  MoveL 2642 to (274.37, 10.03, -264.36) mm, rotated rx -179.9 ry 0 rz -90 deg; joints [33.189, -61.203, 97.914, -131.675, 47.114, 143.425]
  MoveC 2643 to (277.1, 10.02, -263.23) mm, rotated rx -179.9 ry 0 rz -90 deg; joints [33.299, -61.17, 97.861, -131.541, 47.167, 143.324] to (278.23, 10.02, -260.51) mm, rotated rx -179.9 ry 0 rz -90 deg; joints [33.393, -61.271, 98.014, -131.475, 47.257, 143.309]
  MoveL 2644 to (278.23, 10.02, -260.51) mm, rotated rx -179.9 ry 0 rz -90 deg; joints [33.393, -61.271, 98.014, -131.475, 47.257, 143.309]
  MoveL 2645 to (278.23, 10.03, -85.81) mm, rotated rx -179.9 ry 0 rz -90 deg; joints [37.456, -69.808, 110.438, -129.685, 52.193, 144.471]
  MoveC 2646 to (276.95, 10.02, -81.59) mm, rotated rx -179.9 ry 0 rz -90 deg; joints [37.521, -70.054, 110.778, -129.674, 52.292, 144.523] to (273.55, 10.03, -78.79) mm, rotated rx -179.9 ry 0 rz -90 deg; joints [37.48, -70.309, 111.133, -129.777, 52.332, 144.646]
  MoveL 2647 to (273.55, 10.02, -78.79) mm, rotated rx -179.9 ry 0 rz -90 deg; joints [37.48, -70.309, 111.133, -129.777, 52.332, 144.646]
  MoveC 2648 to (270.14, 10.02, -75.98) mm, rotated rx -179.9 ry 0 rz -90 deg; joints [37.438, -70.563, 111.486, -129.878, 52.371, 144.767] to (268.86, 10.02, -71.76) mm, rotated rx -179.9 ry 0 rz -90 deg; joints [37.504, -70.809, 111.823, -129.864, 52.468, 144.816]
  MoveL 2649 to (268.86, 10.02, -71.76) mm, rotated rx -179.9 ry 0 rz -90 deg; joints [37.504, -70.809, 111.823, -129.864, 52.468, 144.816]
  MoveL 2650 to (268.86, 10.02, -61.09) mm, rotated rx -179.9 ry 0 rz -90 deg; joints [37.783, -71.313, 112.509, -129.684, 52.746, 144.821]
  MoveC 2651 to (267.74, 10.03, -58.37) mm, rotated rx -179.9 ry 0 rz -90 deg; joints [37.817, -71.483, 112.74, -129.685, 52.804, 144.86] to (265.01, 10.02, -57.24) mm, rotated rx -179.9 ry 0 rz -90 deg; joints [37.754, -71.635, 112.948, -129.783, 52.804, 144.953]
  MoveL 2652 to (265.01, 10.02, -57.24) mm, rotated rx -179.9 ry 0 rz -90 deg; joints [37.754, -71.635, 112.948, -129.783, 52.804, 144.953]
  MoveL 2653 to (-265.01, 10.02, -57.24) mm, rotated rx -179.9 ry 0 rz -90 deg; joints [15.13, -86.315, 131.2, -158.711, 45.944, 165.304]
  MoveC 2654 to (-267.74, 10.03, -58.37) mm, rotated rx -179.9 ry 0 rz -90 deg; joints [14.976, -86.289, 131.174, -158.919, 45.905, 165.446] to (-268.86, 10.02, -61.09) mm, rotated rx -179.9 ry 0 rz -90 deg; joints [14.882, -86.136, 131.013, -159.043, 45.873, 165.528]
  MoveL 2655 to (-268.86, 10.03, -61.09) mm, rotated rx -179.9 ry 0 rz -90 deg; joints [14.882, -86.136, 131.013, -159.043, 45.873, 165.528]
  MoveL 2656 to (-268.86, 10.02, -251.14) mm, rotated rx -179.9 ry 0 rz -90 deg; joints [12.675, -74.659, 117.443, -161.372, 43.366, 166.653]
  MoveC 2657 to (-267.74, 10.02, -253.87) mm, rotated rx -179.9 ry 0 rz -90 deg; joints [12.698, -74.485, 117.216, -161.322, 43.321, 166.605] to (-265.01, 10.02, -255) mm, rotated rx -179.9 ry 0 rz -90 deg; joints [12.805, -74.383, 117.082, -161.158, 43.316, 166.481]
  MoveL 2658 to (-265.01, 10.03, -255) mm, rotated rx -179.9 ry 0 rz -90 deg; joints [12.805, -74.383, 117.082, -161.158, 43.316, 166.481]
  MoveL 2659 to (265.01, 10.02, -255) mm, rotated rx -179.9 ry 0 rz -90 deg; joints [33.086, -61.986, 99.114, -132.076, 47.331, 143.923]
  MoveC 2660 to (267.74, 10.02, -253.87) mm, rotated rx -179.9 ry 0 rz -90 deg; joints [33.197, -61.954, 99.063, -131.941, 47.384, 143.823] to (268.86, 10.02, -251.14) mm, rotated rx -179.9 ry 0 rz -90 deg; joints [33.291, -62.054, 99.214, -131.873, 47.474, 143.806]
  MoveL 2661 to (268.86, 10.02, -251.14) mm, rotated rx -179.9 ry 0 rz -90 deg; joints [33.291, -62.054, 99.214, -131.873, 47.474, 143.806]
  MoveL 2662 to (268.86, 10.02, -71.76) mm, rotated rx -179.9 ry 0 rz -90 deg; joints [37.504, -70.809, 111.823, -129.864, 52.468, 144.816]
  MoveC 2663 to (266.09, 10.02, -66.2) mm, rotated rx -179.9 ry 0 rz -90 deg; joints [37.555, -71.172, 112.321, -129.89, 52.584, 144.914] to (259.98, 10.02, -65.06) mm, rotated rx -179.9 ry 0 rz -90 deg; joints [37.377, -71.445, 112.699, -130.135, 52.548, 145.124]
  MoveL 2664 to (259.98, 10.03, -65.06) mm, rotated rx -179.9 ry 0 rz -90 deg; joints [37.377, -71.445, 112.699, -130.135, 52.548, 145.124]
  MoveC 2665 to (254.53, 10.03, -66.22) mm, rotated rx -179.9 ry 0 rz -90 deg; joints [37.161, -71.585, 112.895, -130.392, 52.46, 145.31] to (248.97, 10.03, -66.6) mm, rotated rx -179.9 ry 0 rz -90 deg; joints [36.959, -71.764, 113.144, -130.641, 52.391, 145.501]
  MoveL 2666 to (248.97, 10.02, -66.6) mm, rotated rx -179.9 ry 0 rz -90 deg; joints [36.959, -71.764, 113.144, -130.641, 52.391, 145.501]
  MoveL 2667 to (-255.65, 10.03, -66.6) mm, rotated rx -179.9 ry 0 rz -90 deg; joints [15.473, -85.568, 130.397, -158.231, 45.981, 164.961]
  MoveC 2668 to (-258.37, 10.03, -67.73) mm, rotated rx -179.9 ry 0 rz -90 deg; joints [15.321, -85.544, 130.373, -158.436, 45.941, 165.101] to (-259.5, 10.03, -70.46) mm, rotated rx -179.9 ry 0 rz -90 deg; joints [15.226, -85.393, 130.211, -158.559, 45.907, 165.182]
  MoveL 2669 to (-259.5, 10.03, -70.46) mm, rotated rx -179.9 ry 0 rz -90 deg; joints [15.226, -85.393, 130.211, -158.559, 45.907, 165.182]
  MoveL 2670 to (-259.5, 10.03, -241.78) mm, rotated rx -179.9 ry 0 rz -90 deg; joints [13.181, -75.083, 117.987, -160.698, 43.599, 166.199]
  MoveC 2671 to (-258.37, 10.02, -244.5) mm, rotated rx -179.9 ry 0 rz -90 deg; joints [13.203, -74.908, 117.76, -160.65, 43.555, 166.153] to (-255.65, 10.03, -245.63) mm, rotated rx -179.9 ry 0 rz -90 deg; joints [13.31, -74.805, 117.625, -160.488, 43.551, 166.029]
  MoveL 2672 to (-255.65, 10.02, -245.63) mm, rotated rx -179.9 ry 0 rz -90 deg; joints [13.31, -74.805, 117.625, -160.488, 43.551, 166.029]
  MoveL 2673 to (255.65, 10.03, -245.63) mm, rotated rx -179.9 ry 0 rz -90 deg; joints [32.98, -62.765, 100.3, -132.467, 47.543, 144.407]
  MoveC 2674 to (258.37, 10.03, -244.5) mm, rotated rx -179.9 ry 0 rz -90 deg; joints [33.093, -62.734, 100.25, -132.331, 47.596, 144.307] to (259.5, 10.03, -241.78) mm, rotated rx -179.9 ry 0 rz -90 deg; joints [33.187, -62.834, 100.4, -132.261, 47.684, 144.288]
  MoveL 2675 to (259.5, 10.02, -241.78) mm, rotated rx -179.9 ry 0 rz -90 deg; joints [33.187, -62.834, 100.4, -132.261, 47.684, 144.288]
  MoveL 2676 to (259.5, 10.03, -70.46) mm, rotated rx -179.9 ry 0 rz -90 deg; joints [37.22, -71.206, 112.375, -130.248, 52.404, 145.139]
  MoveC 2677 to (258.37, 10.03, -67.73) mm, rotated rx -179.9 ry 0 rz -90 deg; joints [37.253, -71.376, 112.607, -130.251, 52.462, 145.178] to (255.65, 10.02, -66.6) mm, rotated rx -179.9 ry 0 rz -90 deg; joints [37.189, -71.527, 112.815, -130.35, 52.462, 145.272]
  MoveL 2678 to (255.65, 10.03, -66.6) mm, rotated rx -179.9 ry 0 rz -90 deg; joints [37.189, -71.527, 112.815, -130.35, 52.462, 145.272]
  MoveL 2679 to (248.97, 10.02, -66.6) mm, rotated rx -179.9 ry 0 rz -90 deg; joints [36.959, -71.764, 113.144, -130.641, 52.391, 145.501]
  MoveC 2680 to (244.46, 10.03, -67.86) mm, rotated rx -179.9 ry 0 rz -90 deg; joints [36.771, -71.864, 113.283, -130.86, 52.31, 145.656] to (241.27, 10.02, -71.28) mm, rotated rx -179.9 ry 0 rz -90 deg; joints [36.572, -71.812, 113.218, -131.059, 52.188, 145.766]
  MoveL 2681 to (241.27, 10.02, -71.28) mm, rotated rx -179.9 ry 0 rz -90 deg; joints [36.572, -71.812, 113.218, -131.059, 52.188, 145.766]
  MoveC 2682 to (238.08, 10.03, -74.7) mm, rotated rx -179.9 ry 0 rz -90 deg; joints [36.374, -71.76, 113.151, -131.258, 52.067, 145.877] to (233.58, 10.02, -75.96) mm, rotated rx -179.9 ry 0 rz -90 deg; joints [36.185, -71.856, 113.287, -131.479, 51.986, 146.033]
  MoveL 2683 to (233.58, 10.03, -75.96) mm, rotated rx -179.9 ry 0 rz -90 deg; joints [36.185, -71.856, 113.287, -131.479, 51.986, 146.033]
  MoveL 2684 to (-246.29, 10.03, -75.96) mm, rotated rx -179.9 ry 0 rz -90 deg; joints [15.809, -84.825, 129.586, -157.757, 46.008, 164.619]
  MoveC 2685 to (-249.01, 10.02, -77.09) mm, rotated rx -179.9 ry 0 rz -90 deg; joints [15.658, -84.802, 129.563, -157.959, 45.967, 164.757] to (-250.14, 10.03, -79.82) mm, rotated rx -179.9 ry 0 rz -90 deg; joints [15.564, -84.652, 129.401, -158.081, 45.93, 164.836]
  MoveL 2686 to (-250.14, 10.02, -79.82) mm, rotated rx -179.9 ry 0 rz -90 deg; joints [15.564, -84.652, 129.401, -158.081, 45.93, 164.836]
  MoveL 2687 to (-250.14, 10.02, -232.42) mm, rotated rx -179.9 ry 0 rz -90 deg; joints [13.693, -75.502, 118.519, -160.021, 43.832, 165.744]
  MoveC 2688 to (-249.01, 10.02, -235.14) mm, rotated rx -179.9 ry 0 rz -90 deg; joints [13.713, -75.326, 118.294, -159.975, 43.79, 165.699] to (-246.29, 10.02, -236.27) mm, rotated rx -179.9 ry 0 rz -90 deg; joints [13.821, -75.222, 118.158, -159.813, 43.787, 165.577]
  MoveL 2689 to (-246.29, 10.02, -236.27) mm, rotated rx -179.9 ry 0 rz -90 deg; joints [13.821, -75.222, 118.158, -159.813, 43.787, 165.577]
  MoveL 2690 to (246.29, 10.03, -236.27) mm, rotated rx -179.9 ry 0 rz -90 deg; joints [32.873, -63.542, 101.472, -132.85, 47.748, 144.878]
  MoveC 2691 to (249.01, 10.03, -235.14) mm, rotated rx -179.9 ry 0 rz -90 deg; joints [32.987, -63.511, 101.423, -132.713, 47.801, 144.778] to (250.14, 10.03, -232.42) mm, rotated rx -179.9 ry 0 rz -90 deg; joints [33.082, -63.612, 101.571, -132.641, 47.889, 144.757]
  MoveL 2692 to (250.14, 10.03, -232.42) mm, rotated rx -179.9 ry 0 rz -90 deg; joints [33.082, -63.612, 101.571, -132.641, 47.889, 144.757]
  MoveL 2693 to (250.14, 10.03, -79.82) mm, rotated rx -179.9 ry 0 rz -90 deg; joints [36.659, -71.091, 112.231, -130.813, 52.063, 145.458]
  MoveC 2694 to (249.01, 10.03, -77.09) mm, rotated rx -179.9 ry 0 rz -90 deg; joints [36.69, -71.261, 112.464, -130.817, 52.122, 145.499] to (246.29, 10.02, -75.96) mm, rotated rx -179.9 ry 0 rz -90 deg; joints [36.625, -71.411, 112.67, -130.918, 52.122, 145.593]
  MoveL 2695 to (246.29, 10.02, -75.96) mm, rotated rx -179.9 ry 0 rz -90 deg; joints [36.625, -71.411, 112.67, -130.918, 52.122, 145.593]
  MoveL 2696 to (233.58, 10.03, -75.96) mm, rotated rx -179.9 ry 0 rz -90 deg; joints [36.185, -71.856, 113.287, -131.479, 51.986, 146.033]
  MoveC 2697 to (229.36, 10.02, -77.24) mm, rotated rx -179.9 ry 0 rz -90 deg; joints [36.005, -71.941, 113.406, -131.689, 51.908, 146.179] to (226.56, 10.02, -80.65) mm, rotated rx -179.9 ry 0 rz -90 deg; joints [35.82, -71.873, 113.318, -131.872, 51.792, 146.278]
  MoveL 2698 to (226.56, 10.02, -80.65) mm, rotated rx -179.9 ry 0 rz -90 deg; joints [35.82, -71.873, 113.318, -131.872, 51.792, 146.278]
  MoveC 2699 to (223.75, 10.02, -84.05) mm, rotated rx -179.9 ry 0 rz -90 deg; joints [35.636, -71.805, 113.23, -132.055, 51.676, 146.376] to (219.54, 10.03, -85.33) mm, rotated rx -179.9 ry 0 rz -90 deg; joints [35.455, -71.888, 113.346, -132.266, 51.598, 146.524]
  MoveL 2700 to (219.54, 10.03, -85.33) mm, rotated rx -179.9 ry 0 rz -90 deg; joints [35.455, -71.888, 113.346, -132.266, 51.598, 146.524]
  MoveL 2701 to (-236.92, 10.03, -85.33) mm, rotated rx -179.9 ry 0 rz -90 deg; joints [16.137, -84.084, 128.767, -157.288, 46.024, 164.277]
  MoveC 2702 to (-239.65, 10.03, -86.46) mm, rotated rx -179.9 ry 0 rz -90 deg; joints [15.988, -84.063, 128.745, -157.488, 45.983, 164.413] to (-240.78, 10.02, -89.18) mm, rotated rx -179.9 ry 0 rz -90 deg; joints [15.894, -83.915, 128.582, -157.608, 45.944, 164.491]
  MoveL 2703 to (-240.78, 10.02, -89.18) mm, rotated rx -179.9 ry 0 rz -90 deg; joints [15.894, -83.915, 128.582, -157.608, 45.944, 164.491]
  MoveL 2704 to (-240.78, 10.02, -223.05) mm, rotated rx -179.9 ry 0 rz -90 deg; joints [14.21, -75.915, 119.042, -159.339, 44.065, 165.288]
  MoveC 2705 to (-239.65, 10.03, -225.78) mm, rotated rx -179.9 ry 0 rz -90 deg; joints [14.229, -75.739, 118.817, -159.295, 44.024, 165.244] to (-236.92, 10.02, -226.91) mm, rotated rx -179.9 ry 0 rz -90 deg; joints [14.337, -75.634, 118.68, -159.134, 44.023, 165.123]
  MoveL 2706 to (-236.92, 10.02, -226.91) mm, rotated rx -179.9 ry 0 rz -90 deg; joints [14.337, -75.634, 118.68, -159.134, 44.023, 165.123]
  MoveL 2707 to (236.92, 10.02, -226.91) mm, rotated rx -179.9 ry 0 rz -90 deg; joints [32.764, -64.316, 102.631, -133.225, 47.948, 145.336]
  MoveC 2708 to (239.65, 10.02, -225.78) mm, rotated rx -179.9 ry 0 rz -90 deg; joints [32.879, -64.285, 102.582, -133.087, 48.001, 145.236] to (240.78, 10.02, -223.05) mm, rotated rx -179.9 ry 0 rz -90 deg; joints [32.975, -64.386, 102.73, -133.012, 48.088, 145.213]
  MoveL 2709 to (240.78, 10.02, -223.05) mm, rotated rx -179.9 ry 0 rz -90 deg; joints [32.975, -64.386, 102.73, -133.012, 48.088, 145.213]
  MoveL 2710 to (240.78, 10.02, -89.18) mm, rotated rx -179.9 ry 0 rz -90 deg; joints [36.098, -70.969, 112.076, -131.38, 51.724, 145.78]
  MoveC 2711 to (239.65, 10.03, -86.46) mm, rotated rx -179.9 ry 0 rz -90 deg; joints [36.128, -71.139, 112.31, -131.386, 51.783, 145.821] to (236.92, 10.02, -85.33) mm, rotated rx -179.9 ry 0 rz -90 deg; joints [36.063, -71.288, 112.515, -131.488, 51.783, 145.916]
  MoveL 2712 to (236.92, 10.02, -85.33) mm, rotated rx -179.9 ry 0 rz -90 deg; joints [36.063, -71.288, 112.515, -131.488, 51.783, 145.916]
  MoveL 2713 to (219.54, 10.03, -85.33) mm, rotated rx -179.9 ry 0 rz -90 deg; joints [35.455, -71.888, 113.346, -132.266, 51.598, 146.524]
  MoveC 2714 to (215.32, 10.02, -86.61) mm, rotated rx -179.9 ry 0 rz -90 deg; joints [35.275, -71.969, 113.461, -132.477, 51.52, 146.672] to (212.51, 10.03, -90.01) mm, rotated rx -179.9 ry 0 rz -90 deg; joints [35.091, -71.899, 113.369, -132.661, 51.405, 146.771]
  MoveL 2715 to (212.51, 10.03, -90.01) mm, rotated rx -179.9 ry 0 rz -90 deg; joints [35.091, -71.899, 113.369, -132.661, 51.405, 146.771]
  MoveC 2716 to (209.71, 10.03, -93.41) mm, rotated rx -179.9 ry 0 rz -90 deg; joints [34.907, -71.827, 113.276, -132.845, 51.289, 146.871] to (205.49, 10.02, -94.69) mm, rotated rx -179.9 ry 0 rz -90 deg; joints [34.726, -71.906, 113.388, -133.058, 51.212, 147.02]
  MoveL 2717 to (205.49, 10.02, -94.69) mm, rotated rx -179.9 ry 0 rz -90 deg; joints [34.726, -71.906, 113.388, -133.058, 51.212, 147.02]
  MoveL 2718 to (-227.56, 10.02, -94.69) mm, rotated rx -179.9 ry 0 rz -90 deg; joints [16.459, -83.347, 127.939, -156.825, 46.03, 163.935]
  MoveC 2719 to (-230.29, 10.03, -95.82) mm, rotated rx -179.9 ry 0 rz -90 deg; joints [16.311, -83.326, 127.918, -157.022, 45.988, 164.07] to (-231.41, 10.03, -98.54) mm, rotated rx -179.9 ry 0 rz -90 deg; joints [16.218, -83.18, 127.754, -157.14, 45.947, 164.146]
  MoveL 2720 to (-231.41, 10.03, -98.54) mm, rotated rx -179.9 ry 0 rz -90 deg; joints [16.218, -83.18, 127.754, -157.14, 45.947, 164.146]
  MoveL 2721 to (-231.41, 10.02, -213.69) mm, rotated rx -179.9 ry 0 rz -90 deg; joints [14.733, -76.323, 119.554, -158.654, 44.299, 164.831]
  MoveC 2722 to (-230.29, 10.02, -216.42) mm, rotated rx -179.9 ry 0 rz -90 deg; joints [14.751, -76.147, 119.33, -158.611, 44.259, 164.788] to (-227.56, 10.03, -217.54) mm, rotated rx -179.9 ry 0 rz -90 deg; joints [14.858, -76.04, 119.192, -158.451, 44.259, 164.668]
  MoveL 2723 to (-227.56, 10.03, -217.55) mm, rotated rx -179.9 ry 0 rz -90 deg; joints [14.858, -76.04, 119.192, -158.451, 44.259, 164.668]
  MoveL 2724 to (227.56, 10.02, -217.55) mm, rotated rx -179.9 ry 0 rz -90 deg; joints [32.654, -65.088, 103.776, -133.592, 48.142, 145.782]
  MoveC 2725 to (230.29, 10.02, -216.42) mm, rotated rx -179.9 ry 0 rz -90 deg; joints [32.769, -65.058, 103.729, -133.453, 48.195, 145.682] to (231.41, 10.03, -213.69) mm, rotated rx -179.9 ry 0 rz -90 deg; joints [32.866, -65.158, 103.875, -133.376, 48.281, 145.657]
  MoveL 2726 to (231.41, 10.02, -213.69) mm, rotated rx -179.9 ry 0 rz -90 deg; joints [32.866, -65.158, 103.875, -133.376, 48.281, 145.657]
  MoveL 2727 to (231.41, 10.03, -98.54) mm, rotated rx -179.9 ry 0 rz -90 deg; joints [35.54, -70.839, 111.911, -131.948, 51.386, 146.103]
  MoveC 2728 to (230.29, 10.03, -95.82) mm, rotated rx -179.9 ry 0 rz -90 deg; joints [35.569, -71.009, 112.145, -131.955, 51.444, 146.145] to (227.56, 10.03, -94.69) mm, rotated rx -179.9 ry 0 rz -90 deg; joints [35.502, -71.158, 112.35, -132.059, 51.445, 146.241]
  MoveL 2729 to (227.56, 10.03, -94.69) mm, rotated rx -179.9 ry 0 rz -90 deg; joints [35.502, -71.158, 112.35, -132.059, 51.445, 146.241]
  MoveL 2730 to (205.49, 10.02, -94.69) mm, rotated rx -179.9 ry 0 rz -90 deg; joints [34.726, -71.906, 113.388, -133.058, 51.212, 147.02]
  MoveC 2731 to (201.27, 10.02, -95.97) mm, rotated rx -179.9 ry 0 rz -90 deg; joints [34.544, -71.985, 113.499, -133.273, 51.134, 147.17] to (198.47, 10.03, -99.37) mm, rotated rx -179.9 ry 0 rz -90 deg; joints [34.361, -71.911, 113.403, -133.457, 51.019, 147.27]
  MoveL 2732 to (198.47, 10.02, -99.37) mm, rotated rx -179.9 ry 0 rz -90 deg; joints [34.361, -71.911, 113.403, -133.457, 51.019, 147.27]
  MoveC 2733 to (195.67, 10.02, -102.78) mm, rotated rx -179.9 ry 0 rz -90 deg; joints [34.177, -71.836, 113.305, -133.642, 50.904, 147.371] to (191.45, 10.02, -104.05) mm, rotated rx -179.9 ry 0 rz -90 deg; joints [33.995, -71.912, 113.413, -133.858, 50.827, 147.521]
  MoveL 2734 to (191.45, 10.02, -104.05) mm, rotated rx -179.9 ry 0 rz -90 deg; joints [33.995, -71.912, 113.413, -133.858, 50.827, 147.521]
  MoveL 2735 to (-218.2, 10.02, -104.05) mm, rotated rx -179.9 ry 0 rz -90 deg; joints [16.775, -82.612, 127.102, -156.366, 46.027, 163.592]
  MoveC 2736 to (-220.92, 10.02, -105.18) mm, rotated rx -179.9 ry 0 rz -90 deg; joints [16.628, -82.592, 127.082, -156.561, 45.984, 163.725] to (-222.05, 10.02, -107.91) mm, rotated rx -179.9 ry 0 rz -90 deg; joints [16.535, -82.448, 126.918, -156.677, 45.94, 163.8]
  MoveL 2737 to (-222.05, 10.03, -107.91) mm, rotated rx -179.9 ry 0 rz -90 deg; joints [16.535, -82.448, 126.918, -156.677, 45.94, 163.8]
  MoveL 2738 to (-222.05, 10.02, -204.33) mm, rotated rx -179.9 ry 0 rz -90 deg; joints [15.261, -76.726, 120.056, -157.964, 44.534, 164.373]
  MoveC 2739 to (-220.92, 10.03, -207.05) mm, rotated rx -179.9 ry 0 rz -90 deg; joints [15.278, -76.549, 119.833, -157.923, 44.495, 164.331] to (-218.2, 10.02, -208.18) mm, rotated rx -179.9 ry 0 rz -90 deg; joints [15.385, -76.44, 119.693, -157.765, 44.496, 164.212]
  MoveL 2740 to (-218.2, 10.03, -208.18) mm, rotated rx -179.9 ry 0 rz -90 deg; joints [15.385, -76.44, 119.693, -157.765, 44.496, 164.212]
  MoveL 2741 to (218.2, 10.03, -208.18) mm, rotated rx -179.9 ry 0 rz -90 deg; joints [32.541, -65.858, 104.909, -133.951, 48.329, 146.215]
  MoveC 2742 to (220.92, 10.02, -207.05) mm, rotated rx -179.9 ry 0 rz -90 deg; joints [32.657, -65.828, 104.863, -133.811, 48.383, 146.115] to (222.05, 10.02, -204.33) mm, rotated rx -179.9 ry 0 rz -90 deg; joints [32.755, -65.929, 105.008, -133.732, 48.468, 146.088]
  MoveL 2743 to (222.05, 10.02, -204.33) mm, rotated rx -179.9 ry 0 rz -90 deg; joints [32.755, -65.929, 105.008, -133.732, 48.468, 146.088]
  MoveL 2744 to (222.05, 10.02, -107.91) mm, rotated rx -179.9 ry 0 rz -90 deg; joints [34.983, -70.701, 111.734, -132.517, 51.049, 146.428]
  MoveC 2745 to (220.92, 10.02, -105.18) mm, rotated rx -179.9 ry 0 rz -90 deg; joints [35.011, -70.872, 111.969, -132.526, 51.107, 146.47] to (218.2, 10.02, -104.05) mm, rotated rx -179.9 ry 0 rz -90 deg; joints [34.943, -71.02, 112.173, -132.632, 51.108, 146.568]
  MoveL 2746 to (218.2, 10.02, -104.05) mm, rotated rx -179.9 ry 0 rz -90 deg; joints [34.943, -71.02, 112.173, -132.632, 51.108, 146.568]
  MoveL 2747 to (191.45, 10.02, -104.05) mm, rotated rx -179.9 ry 0 rz -90 deg; joints [33.995, -71.912, 113.413, -133.858, 50.827, 147.521]
  MoveC 2748 to (187.23, 10.03, -105.33) mm, rotated rx -179.9 ry 0 rz -90 deg; joints [33.813, -71.988, 113.519, -134.074, 50.751, 147.672] to (184.43, 10.02, -108.73) mm, rotated rx -179.9 ry 0 rz -90 deg; joints [33.63, -71.911, 113.419, -134.26, 50.636, 147.774]
  MoveL 2749 to (184.43, 10.02, -108.73) mm, rotated rx -179.9 ry 0 rz -90 deg; joints [33.63, -71.911, 113.419, -134.26, 50.636, 147.774]
  MoveC 2750 to (181.62, 10.02, -112.14) mm, rotated rx -179.9 ry 0 rz -90 deg; joints [33.448, -71.832, 113.317, -134.445, 50.522, 147.876] to (177.4, 10.02, -113.42) mm, rotated rx -179.9 ry 0 rz -90 deg; joints [33.265, -71.906, 113.42, -134.663, 50.446, 148.028]
  MoveL 2751 to (177.4, 10.02, -113.42) mm, rotated rx -179.9 ry 0 rz -90 deg; joints [33.265, -71.906, 113.42, -134.663, 50.446, 148.028]
  MoveL 2752 to (-208.84, 10.02, -113.42) mm, rotated rx -179.9 ry 0 rz -90 deg; joints [17.084, -81.879, 126.257, -155.911, 46.013, 163.249]
  MoveC 2753 to (-211.56, 10.03, -114.54) mm, rotated rx -179.9 ry 0 rz -90 deg; joints [16.938, -81.861, 126.238, -156.104, 45.97, 163.38] to (-212.69, 10.03, -117.27) mm, rotated rx -179.9 ry 0 rz -90 deg; joints [16.846, -81.718, 126.074, -156.219, 45.924, 163.453]
  MoveL 2754 to (-212.69, 10.03, -117.27) mm, rotated rx -179.9 ry 0 rz -90 deg; joints [16.846, -81.718, 126.074, -156.219, 45.924, 163.453]
  MoveL 2755 to (-212.69, 10.03, -194.97) mm, rotated rx -179.9 ry 0 rz -90 deg; joints [15.795, -77.123, 120.548, -157.271, 44.769, 163.913]
  MoveC 2756 to (-211.56, 10.02, -197.69) mm, rotated rx -179.9 ry 0 rz -90 deg; joints [15.811, -76.946, 120.325, -157.231, 44.731, 163.873] to (-208.84, 10.02, -198.82) mm, rotated rx -179.9 ry 0 rz -90 deg; joints [15.918, -76.835, 120.184, -157.074, 44.734, 163.755]
  MoveL 2757 to (-208.84, 10.03, -198.82) mm, rotated rx -179.9 ry 0 rz -90 deg; joints [15.918, -76.835, 120.184, -157.074, 44.734, 163.755]
  MoveL 2758 to (208.84, 10.03, -198.82) mm, rotated rx -179.9 ry 0 rz -90 deg; joints [32.426, -66.626, 106.03, -134.303, 48.511, 146.636]
  MoveC 2759 to (211.56, 10.02, -197.69) mm, rotated rx -179.9 ry 0 rz -90 deg; joints [32.543, -66.596, 105.984, -134.162, 48.565, 146.536] to (212.69, 10.02, -194.97) mm, rotated rx -179.9 ry 0 rz -90 deg; joints [32.641, -66.697, 106.129, -134.081, 48.649, 146.507]
  MoveL 2760 to (212.69, 10.03, -194.97) mm, rotated rx -179.9 ry 0 rz -90 deg; joints [32.641, -66.697, 106.129, -134.081, 48.649, 146.507]
  MoveL 2761 to (212.69, 10.02, -117.27) mm, rotated rx -179.9 ry 0 rz -90 deg; joints [34.429, -70.556, 111.547, -133.087, 50.713, 146.755]
  MoveC 2762 to (211.56, 10.03, -114.54) mm, rotated rx -179.9 ry 0 rz -90 deg; joints [34.455, -70.728, 111.783, -133.097, 50.772, 146.798] to (208.84, 10.03, -113.42) mm, rotated rx -179.9 ry 0 rz -90 deg; joints [34.386, -70.874, 111.986, -133.205, 50.773, 146.897]
  MoveL 2763 to (208.84, 10.03, -113.42) mm, rotated rx -179.9 ry 0 rz -90 deg; joints [34.386, -70.874, 111.986, -133.205, 50.773, 146.897]
  MoveL 2764 to (177.4, 10.02, -113.42) mm, rotated rx -179.9 ry 0 rz -90 deg; joints [33.265, -71.906, 113.42, -134.663, 50.446, 148.028]
  MoveC 2765 to (173.18, 10.03, -114.69) mm, rotated rx -179.9 ry 0 rz -90 deg; joints [33.082, -71.978, 113.522, -134.882, 50.369, 148.181] to (170.38, 10.03, -118.1) mm, rotated rx -179.9 ry 0 rz -90 deg; joints [32.9, -71.897, 113.417, -135.068, 50.255, 148.283]
  MoveL 2766 to (170.38, 10.03, -118.1) mm, rotated rx -179.9 ry 0 rz -90 deg; joints [32.9, -71.897, 113.417, -135.068, 50.255, 148.283]
  MoveC 2767 to (167.58, 10.02, -121.5) mm, rotated rx -179.9 ry 0 rz -90 deg; joints [32.718, -71.816, 113.311, -135.254, 50.142, 148.386] to (163.36, 10.02, -122.78) mm, rotated rx -179.9 ry 0 rz -90 deg; joints [32.535, -71.886, 113.41, -135.474, 50.066, 148.54]
  MoveL 2768 to (163.36, 10.02, -122.78) mm, rotated rx -179.9 ry 0 rz -90 deg; joints [32.535, -71.886, 113.41, -135.474, 50.066, 148.54]
  MoveL 2769 to (-199.47, 10.02, -122.78) mm, rotated rx -179.9 ry 0 rz -90 deg; joints [17.386, -81.149, 125.404, -155.459, 45.99, 162.904]
  MoveC 2770 to (-202.2, 10.03, -123.91) mm, rotated rx -179.9 ry 0 rz -90 deg; joints [17.243, -81.131, 125.385, -155.65, 45.946, 163.034] to (-203.33, 10.03, -126.63) mm, rotated rx -179.9 ry 0 rz -90 deg; joints [17.15, -80.99, 125.221, -155.764, 45.898, 163.104]
  MoveL 2771 to (-203.33, 10.03, -126.63) mm, rotated rx -179.9 ry 0 rz -90 deg; joints [17.15, -80.99, 125.221, -155.764, 45.898, 163.104]
  MoveL 2772 to (-203.33, 10.02, -185.6) mm, rotated rx -179.9 ry 0 rz -90 deg; joints [16.335, -77.515, 121.029, -156.573, 45.005, 163.452]
  MoveC 2773 to (-202.2, 10.03, -188.33) mm, rotated rx -179.9 ry 0 rz -90 deg; joints [16.349, -77.337, 120.807, -156.536, 44.968, 163.414] to (-199.47, 10.02, -189.46) mm, rotated rx -179.9 ry 0 rz -90 deg; joints [16.456, -77.225, 120.665, -156.38, 44.972, 163.297]
  MoveL 2774 to (-199.47, 10.02, -189.46) mm, rotated rx -179.9 ry 0 rz -90 deg; joints [16.456, -77.225, 120.665, -156.38, 44.972, 163.297]
  MoveL 2775 to (199.47, 10.03, -189.46) mm, rotated rx -179.9 ry 0 rz -90 deg; joints [32.308, -67.393, 107.139, -134.649, 48.686, 147.046]
  MoveC 2776 to (202.2, 10.03, -188.33) mm, rotated rx -179.9 ry 0 rz -90 deg; joints [32.427, -67.364, 107.094, -134.507, 48.74, 146.946] to (203.33, 10.03, -185.6) mm, rotated rx -179.9 ry 0 rz -90 deg; joints [32.526, -67.465, 107.237, -134.423, 48.824, 146.915]
  MoveL 2777 to (203.33, 10.02, -185.6) mm, rotated rx -179.9 ry 0 rz -90 deg; joints [32.526, -67.465, 107.237, -134.423, 48.824, 146.915]
  MoveL 2778 to (203.33, 10.03, -126.63) mm, rotated rx -179.9 ry 0 rz -90 deg; joints [33.876, -70.404, 111.349, -133.658, 50.379, 147.083]
  MoveC 2779 to (202.2, 10.03, -123.91) mm, rotated rx -179.9 ry 0 rz -90 deg; joints [33.901, -70.576, 111.586, -133.67, 50.437, 147.127] to (199.47, 10.03, -122.78) mm, rotated rx -179.9 ry 0 rz -90 deg; joints [33.831, -70.721, 111.788, -133.779, 50.438, 147.227]
  MoveL 2780 to (199.47, 10.03, -122.78) mm, rotated rx -179.9 ry 0 rz -90 deg; joints [33.831, -70.721, 111.788, -133.779, 50.438, 147.227]
  MoveL 2781 to (163.36, 10.02, -122.78) mm, rotated rx -179.9 ry 0 rz -90 deg; joints [32.535, -71.886, 113.41, -135.474, 50.066, 148.54]
  MoveC 2782 to (159.14, 10.02, -124.06) mm, rotated rx -179.9 ry 0 rz -90 deg; joints [32.351, -71.955, 113.508, -135.695, 49.99, 148.694] to (156.34, 10.03, -127.46) mm, rotated rx -179.9 ry 0 rz -90 deg; joints [32.17, -71.872, 113.398, -135.882, 49.877, 148.798]
  MoveL 2783 to (156.34, 10.03, -127.46) mm, rotated rx -179.9 ry 0 rz -90 deg; joints [32.17, -71.872, 113.398, -135.882, 49.877, 148.798]
  MoveC 2784 to (153.54, 10.02, -130.86) mm, rotated rx -179.9 ry 0 rz -90 deg; joints [31.989, -71.787, 113.288, -136.069, 49.764, 148.901] to (149.32, 10.03, -132.14) mm, rotated rx -179.9 ry 0 rz -90 deg; joints [31.805, -71.854, 113.382, -136.291, 49.689, 149.057]
  MoveL 2785 to (149.32, 10.03, -132.14) mm, rotated rx -179.9 ry 0 rz -90 deg; joints [31.805, -71.854, 113.382, -136.291, 49.689, 149.057]
  MoveL 2786 to (-190.11, 10.03, -132.14) mm, rotated rx -179.9 ry 0 rz -90 deg; joints [17.683, -80.421, 124.541, -155.011, 45.957, 162.557]
  MoveC 2787 to (-192.84, 10.03, -133.27) mm, rotated rx -179.9 ry 0 rz -90 deg; joints [17.541, -80.404, 124.524, -155.2, 45.913, 162.685] to (-193.96, 10.02, -135.99) mm, rotated rx -179.9 ry 0 rz -90 deg; joints [17.449, -80.264, 124.359, -155.312, 45.863, 162.754]
  MoveL 2788 to (-193.96, 10.02, -135.99) mm, rotated rx -179.9 ry 0 rz -90 deg; joints [17.449, -80.264, 124.359, -155.312, 45.863, 162.754]
  MoveL 2789 to (-193.96, 10.02, -176.24) mm, rotated rx -179.9 ry 0 rz -90 deg; joints [16.88, -77.901, 121.5, -155.871, 45.242, 162.991]
  MoveC 2790 to (-192.84, 10.02, -178.97) mm, rotated rx -179.9 ry 0 rz -90 deg; joints [16.893, -77.722, 121.278, -155.836, 45.207, 162.954] to (-190.11, 10.02, -180.09) mm, rotated rx -179.9 ry 0 rz -90 deg; joints [17, -77.609, 121.136, -155.681, 45.212, 162.838]
  MoveL 2791 to (-190.11, 10.02, -180.09) mm, rotated rx -179.9 ry 0 rz -90 deg; joints [17, -77.609, 121.136, -155.681, 45.212, 162.838]
  MoveL 2792 to (190.11, 10.03, -180.09) mm, rotated rx -179.9 ry 0 rz -90 deg; joints [32.189, -68.159, 108.236, -134.988, 48.855, 147.444]
  MoveC 2793 to (192.84, 10.02, -178.97) mm, rotated rx -179.9 ry 0 rz -90 deg; joints [32.309, -68.13, 108.193, -134.845, 48.909, 147.344] to (193.96, 10.02, -176.24) mm, rotated rx -179.9 ry 0 rz -90 deg; joints [32.409, -68.231, 108.335, -134.759, 48.992, 147.311]
  MoveL 2794 to (193.96, 10.03, -176.24) mm, rotated rx -179.9 ry 0 rz -90 deg; joints [32.409, -68.231, 108.335, -134.759, 48.992, 147.311]
  MoveL 2795 to (193.96, 10.02, -135.99) mm, rotated rx -179.9 ry 0 rz -90 deg; joints [33.325, -70.244, 111.141, -134.23, 50.045, 147.413]
  MoveC 2796 to (192.84, 10.02, -133.27) mm, rotated rx -179.9 ry 0 rz -90 deg; joints [33.349, -70.416, 111.379, -134.243, 50.104, 147.458] to (190.11, 10.02, -132.14) mm, rotated rx -179.9 ry 0 rz -90 deg; joints [33.279, -70.561, 111.58, -134.354, 50.105, 147.559]
  MoveL 2797 to (190.11, 10.03, -132.14) mm, rotated rx -179.9 ry 0 rz -90 deg; joints [33.279, -70.561, 111.58, -134.354, 50.105, 147.559]
  MoveL 2798 to (149.32, 10.03, -132.14) mm, rotated rx -179.9 ry 0 rz -90 deg; joints [31.805, -71.854, 113.382, -136.291, 49.689, 149.057]
  MoveC 2799 to (145.1, 10.02, -133.42) mm, rotated rx -179.9 ry 0 rz -90 deg; joints [31.621, -71.92, 113.476, -136.515, 49.614, 149.213] to (142.29, 10.02, -136.82) mm, rotated rx -179.9 ry 0 rz -90 deg; joints [31.44, -71.833, 113.362, -136.702, 49.501, 149.317]
  MoveL 2800 to (142.29, 10.03, -136.82) mm, rotated rx -179.9 ry 0 rz -90 deg; joints [31.44, -71.833, 113.362, -136.702, 49.501, 149.317]
  MoveC 2801 to (139.49, 10.03, -140.23) mm, rotated rx -179.9 ry 0 rz -90 deg; joints [31.26, -71.746, 113.247, -136.889, 49.389, 149.422] to (135.27, 10.02, -141.5) mm, rotated rx -179.9 ry 0 rz -90 deg; joints [31.076, -71.809, 113.337, -137.114, 49.314, 149.579]
  MoveL 2802 to (135.27, 10.02, -141.5) mm, rotated rx -179.9 ry 0 rz -90 deg; joints [31.076, -71.809, 113.337, -137.114, 49.314, 149.579]
  MoveL 2803 to (-180.75, 10.03, -141.5) mm, rotated rx -179.9 ry 0 rz -90 deg; joints [17.974, -79.694, 123.67, -154.566, 45.915, 162.208]
  MoveC 2804 to (-183.47, 10.02, -142.63) mm, rotated rx -179.9 ry 0 rz -90 deg; joints [17.833, -79.679, 123.654, -154.753, 45.871, 162.335] to (-184.6, 10.03, -145.36) mm, rotated rx -179.9 ry 0 rz -90 deg; joints [17.741, -79.54, 123.488, -154.863, 45.819, 162.402]
  MoveL 2805 to (-184.6, 10.03, -145.36) mm, rotated rx -179.9 ry 0 rz -90 deg; joints [17.741, -79.54, 123.488, -154.863, 45.819, 162.402]
  MoveL 2806 to (-184.6, 10.02, -166.88) mm, rotated rx -179.9 ry 0 rz -90 deg; joints [17.431, -78.281, 121.96, -155.166, 45.481, 162.528]
  MoveC 2807 to (-183.47, 10.02, -169.6) mm, rotated rx -179.9 ry 0 rz -90 deg; joints [17.443, -78.101, 121.74, -155.133, 45.446, 162.492] to (-180.75, 10.02, -170.73) mm, rotated rx -179.9 ry 0 rz -90 deg; joints [17.549, -77.986, 121.596, -154.979, 45.453, 162.378]
  MoveL 2808 to (-180.75, 10.02, -170.73) mm, rotated rx -179.9 ry 0 rz -90 deg; joints [17.549, -77.986, 121.596, -154.979, 45.453, 162.378]
  MoveL 2809 to (180.75, 10.03, -170.73) mm, rotated rx -179.9 ry 0 rz -90 deg; joints [32.068, -68.924, 109.323, -135.321, 49.017, 147.832]
  MoveC 2810 to (183.47, 10.02, -169.6) mm, rotated rx -179.9 ry 0 rz -90 deg; joints [32.189, -68.895, 109.28, -135.177, 49.072, 147.732] to (184.6, 10.02, -166.88) mm, rotated rx -179.9 ry 0 rz -90 deg; joints [32.289, -68.997, 109.421, -135.089, 49.154, 147.697]
  MoveL 2811 to (184.6, 10.02, -166.88) mm, rotated rx -179.9 ry 0 rz -90 deg; joints [32.289, -68.997, 109.421, -135.089, 49.154, 147.697]
  MoveL 2812 to (184.6, 10.02, -145.36) mm, rotated rx -179.9 ry 0 rz -90 deg; joints [32.777, -70.077, 110.921, -134.802, 49.712, 147.744]
  MoveC 2813 to (183.47, 10.02, -142.63) mm, rotated rx -179.9 ry 0 rz -90 deg; joints [32.799, -70.25, 111.16, -134.817, 49.771, 147.79] to (180.75, 10.02, -141.5) mm, rotated rx -179.9 ry 0 rz -90 deg; joints [32.728, -70.393, 111.36, -134.93, 49.773, 147.893]
  MoveL 2814 to (180.75, 10.02, -141.5) mm, rotated rx -179.9 ry 0 rz -90 deg; joints [32.728, -70.393, 111.36, -134.93, 49.773, 147.893]
  MoveL 2815 to (135.27, 10.02, -141.5) mm, rotated rx -179.9 ry 0 rz -90 deg; joints [31.076, -71.809, 113.337, -137.114, 49.314, 149.579]
  MoveC 2816 to (131.05, 10.02, -142.78) mm, rotated rx -179.9 ry 0 rz -90 deg; joints [30.891, -71.872, 113.426, -137.339, 49.24, 149.737] to (128.25, 10.02, -146.18) mm, rotated rx -179.9 ry 0 rz -90 deg; joints [30.711, -71.782, 113.308, -137.527, 49.128, 149.842]
  MoveL 2817 to (128.25, 10.02, -146.18) mm, rotated rx -179.9 ry 0 rz -90 deg; joints [30.711, -71.782, 113.308, -137.527, 49.128, 149.842]
  MoveC 2818 to (125.45, 10.02, -149.59) mm, rotated rx -179.9 ry 0 rz -90 deg; joints [30.532, -71.691, 113.189, -137.715, 49.016, 149.948] to (121.23, 10.02, -150.87) mm, rotated rx -179.9 ry 0 rz -90 deg; joints [30.347, -71.752, 113.275, -137.942, 48.942, 150.107]
  MoveL 2819 to (121.23, 10.03, -150.87) mm, rotated rx -179.9 ry 0 rz -90 deg; joints [30.347, -71.752, 113.275, -137.942, 48.942, 150.107]
  MoveL 2820 to (-171.39, 10.03, -150.87) mm, rotated rx -179.9 ry 0 rz -90 deg; joints [18.26, -78.97, 122.791, -154.124, 45.865, 161.856]
  MoveC 2821 to (-174.11, 10.02, -151.99) mm, rotated rx -179.9 ry 0 rz -90 deg; joints [18.12, -78.955, 122.776, -154.308, 45.82, 161.982] to (-175.24, 10.02, -154.72) mm, rotated rx -179.9 ry 0 rz -90 deg; joints [18.028, -78.818, 122.609, -154.417, 45.765, 162.048]
  MoveL 2822 to (-175.24, 10.02, -154.72) mm, rotated rx -179.9 ry 0 rz -90 deg; joints [18.028, -78.818, 122.609, -154.417, 45.765, 162.048]
  MoveL 2823 to (-175.24, 10.02, -157.52) mm, rotated rx -179.9 ry 0 rz -90 deg; joints [17.987, -78.655, 122.411, -154.457, 45.721, 162.064]
  MoveC 2824 to (-174.11, 10.02, -160.24) mm, rotated rx -179.9 ry 0 rz -90 deg; joints [17.998, -78.475, 122.191, -154.426, 45.688, 162.03] to (-171.39, 10.03, -161.37) mm, rotated rx -179.9 ry 0 rz -90 deg; joints [18.104, -78.358, 122.046, -154.274, 45.695, 161.917]
  MoveL 2825 to (-171.39, 10.02, -161.37) mm, rotated rx -179.9 ry 0 rz -90 deg; joints [18.104, -78.358, 122.046, -154.274, 45.695, 161.917]
  MoveL 2826 to (171.39, 10.02, -161.37) mm, rotated rx -179.9 ry 0 rz -90 deg; joints [31.944, -69.688, 110.398, -135.649, 49.173, 148.209]
  MoveC 2827 to (174.11, 10.02, -160.24) mm, rotated rx -179.9 ry 0 rz -90 deg; joints [32.066, -69.66, 110.356, -135.503, 49.228, 148.109] to (175.24, 10.02, -157.52) mm, rotated rx -179.9 ry 0 rz -90 deg; joints [32.167, -69.762, 110.496, -135.413, 49.309, 148.072]
  MoveL 2828 to (175.24, 10.03, -157.52) mm, rotated rx -179.9 ry 0 rz -90 deg; joints [32.167, -69.762, 110.496, -135.413, 49.309, 148.072]
  MoveL 2829 to (175.24, 10.02, -154.72) mm, rotated rx -179.9 ry 0 rz -90 deg; joints [32.23, -69.903, 110.691, -135.376, 49.381, 148.077]
  MoveC 2830 to (174.11, 10.03, -151.99) mm, rotated rx -179.9 ry 0 rz -90 deg; joints [32.252, -70.076, 110.931, -135.392, 49.44, 148.124] to (171.39, 10.03, -150.87) mm, rotated rx -179.9 ry 0 rz -90 deg; joints [32.18, -70.218, 111.13, -135.507, 49.442, 148.228]
  MoveL 2831 to (171.39, 10.02, -150.87) mm, rotated rx -179.9 ry 0 rz -90 deg; joints [32.18, -70.218, 111.13, -135.507, 49.442, 148.228]
  MoveL 2832 to (121.23, 10.03, -150.87) mm, rotated rx -179.9 ry 0 rz -90 deg; joints [30.347, -71.752, 113.275, -137.942, 48.942, 150.107]
  MoveL 2833 to (121.01, 10.04, -150.88) mm, rotated rx -179.9 ry 0 rz -90 deg; joints [30.339, -71.758, 113.282, -137.953, 48.939, 150.114]
  MoveL 2834 to (120.8, 10.1, -150.94) mm, rotated rx -179.9 ry 0 rz -90 deg; joints [30.33, -71.763, 113.285, -137.961, 48.932, 150.118]
  MoveL 2835 to (120.62, 10.2, -151.02) mm, rotated rx -179.9 ry 0 rz -90 deg; joints [30.321, -71.768, 113.284, -137.968, 48.924, 150.12]
  MoveL 2836 to (120.47, 10.32, -151.12) mm, rotated rx -179.9 ry 0 rz -90 deg; joints [30.313, -71.772, 113.279, -137.972, 48.913, 150.118]
  MoveL 2837 to (120.35, 10.48, -151.22) mm, rotated rx -179.9 ry 0 rz -90 deg; joints [30.307, -71.776, 113.272, -137.973, 48.902, 150.113]
  MoveL 2838 to (120.26, 10.66, -151.31) mm, rotated rx -179.9 ry 0 rz -90 deg; joints [30.301, -71.78, 113.263, -137.972, 48.89, 150.105]
  MoveL 2839 to (120.2, 10.86, -151.39) mm, rotated rx -179.9 ry 0 rz -90 deg; joints [30.297, -71.785, 113.254, -137.968, 48.877, 150.096]
  MoveL 2840 to (120.17, 11.07, -151.43) mm, rotated rx -179.9 ry 0 rz -90 deg; joints [30.295, -71.791, 113.245, -137.962, 48.865, 150.084]
  MoveL 2841 to (120.16, 11.29, -151.45) mm, rotated rx -179.9 ry 0 rz -90 deg; joints [30.294, -71.798, 113.238, -137.954, 48.853, 150.071]
  Set speed (1000.0 mm/s)
  MoveL 2842 to (120.16, 110.53, -151.45) mm, rotated rx -179.9 ry 0 rz -90 deg; joints [30.245, -74.935, 109.673, -133.558, 44.02, 143.657]
  MoveL 2843 to (325.1, 110.53, -224.13) mm, rotated rx -179.9 ry 0 rz -90 deg; joints [35.606, -64.15, 94.756, -124.49, 44.928, 135.019]
  Set speed (100.0 mm/s)
  MoveL 2844 to (325.1, 37.54, -224.13) mm, rotated rx -179.9 ry 0 rz -90 deg; joints [35.641, -62.287, 97.412, -127.944, 47.624, 140.04]
  MoveC 2845 to (325.1, 36.66, -224.48) mm, rotated rx -179.9 ry 0 rz -90 deg; joints [35.634, -62.244, 97.414, -127.984, 47.647, 140.093] to (325.1, 36.27, -225.35) mm, rotated rx -179.9 ry 0 rz -90 deg; joints [35.614, -62.19, 97.362, -128.006, 47.636, 140.109]
  MoveL 2846 to (325.1, 36.27, -225.35) mm, rotated rx -179.9 ry 0 rz -90 deg; joints [35.614, -62.19, 97.362, -128.006, 47.636, 140.109]
  MoveL 2847 to (325.1, 33.28, -311.23) mm, rotated rx -179.9 ry 0 rz -90 deg; joints [33.788, -57.704, 90.697, -128.287, 45.1, 139.032]
  MoveL 2848 to (322.43, 33.18, -311.23) mm, rotated rx -179.9 ry 0 rz -90 deg; joints [33.706, -57.795, 90.849, -128.421, 45.085, 139.16]
  MoveL 2849 to (322.43, 22.35, -1) mm, rotated rx -179.9 ry 0 rz -90 deg; joints [41.207, -72.507, 113.061, -125.898, 54.399, 142.22]
  MoveL 2850 to (325.1, 22.26, -1) mm, rotated rx -179.9 ry 0 rz -90 deg; joints [41.294, -72.398, 112.921, -125.795, 54.434, 142.141]
  MoveL 2851 to (325.1, 11.42, -311.23) mm, rotated rx -179.9 ry 0 rz -90 deg; joints [33.797, -57.123, 91.407, -129.266, 45.915, 140.437]
  MoveL 2852 to (322.43, 11.33, -311.23) mm, rotated rx -179.9 ry 0 rz -90 deg; joints [33.716, -57.212, 91.559, -129.399, 45.903, 140.563]
  MoveL 2853 to (322.43, 0.5, -1.13) mm, rotated rx -179.9 ry 0 rz -90 deg; joints [41.216, -71.728, 113.755, -126.725, 55.277, 143.667]
  MoveL 2854 to (322.43, 0.5, -1) mm, rotated rx -179.9 ry 0 rz -90 deg; joints [41.22, -71.734, 113.763, -126.723, 55.28, 143.667]
  MoveL 2855 to (325.1, 0.5, -1) mm, rotated rx -179.9 ry 0 rz -90 deg; joints [41.307, -71.63, 113.619, -126.616, 55.308, 143.581]
  MoveL 2856 to (325.1, 0.5, -311.23) mm, rotated rx -179.9 ry 0 rz -90 deg; joints [33.802, -56.821, 91.747, -129.737, 46.327, 141.12]
  MoveL 2857 to (322.43, 0.5, -311.23) mm, rotated rx -179.9 ry 0 rz -90 deg; joints [33.721, -56.913, 91.896, -129.866, 46.312, 141.24]
  MoveL 2858 to (322.43, 0.5, -1.13) mm, rotated rx -179.9 ry 0 rz -90 deg; joints [41.216, -71.728, 113.755, -126.725, 55.277, 143.667]
  MoveL 2859 to (322.43, 1.77, -1.13) mm, rotated rx -179.9 ry 0 rz -90 deg; joints [41.216, -71.774, 113.715, -126.678, 55.225, 143.584]
  Set speed (1000.0 mm/s)
  MoveL 2860 to (322.43, 110.53, -1.13) mm, rotated rx -179.9 ry 0 rz -90 deg; joints [41.152, -75.252, 109.839, -122.181, 51.019, 136.036]
  MoveL 2861 to (-319.75, 110.53, -6.58) mm, rotated rx -179.9 ry 0 rz -90 deg; joints [12.881, -94.526, 131.236, -158.634, 37.709, 163.228]
  Set speed (100.0 mm/s)
  MoveL 2862 to (-319.75, 37.54, -6.58) mm, rotated rx -179.9 ry 0 rz -90 deg; joints [12.911, -91.707, 134.377, -160.999, 43.313, 166.36]
  MoveL 2863 to (-319.73, 37.33, -6.58) mm, rotated rx -179.9 ry 0 rz -90 deg; joints [12.912, -91.698, 134.386, -161.004, 43.331, 166.368]
  MoveL 2864 to (-319.68, 37.12, -6.56) mm, rotated rx -179.9 ry 0 rz -90 deg; joints [12.915, -91.689, 134.395, -161.005, 43.348, 166.373]
  MoveL 2865 to (-319.6, 36.92, -6.53) mm, rotated rx -179.9 ry 0 rz -90 deg; joints [12.92, -91.682, 134.404, -161.004, 43.364, 166.375]
  MoveL 2866 to (-319.48, 36.74, -6.49) mm, rotated rx -179.9 ry 0 rz -90 deg; joints [12.927, -91.675, 134.412, -160.999, 43.38, 166.375]
  MoveL 2867 to (-319.34, 36.59, -6.44) mm, rotated rx -179.9 ry 0 rz -90 deg; joints [12.935, -91.669, 134.419, -160.992, 43.394, 166.373]
  MoveL 2868 to (-319.17, 36.46, -6.39) mm, rotated rx -179.9 ry 0 rz -90 deg; joints [12.945, -91.665, 134.425, -160.982, 43.407, 166.368]
  MoveL 2869 to (-318.98, 36.36, -6.34) mm, rotated rx -179.9 ry 0 rz -90 deg; joints [12.956, -91.661, 134.429, -160.969, 43.417, 166.361]
  MoveL 2870 to (-318.78, 36.3, -6.29) mm, rotated rx -179.9 ry 0 rz -90 deg; joints [12.968, -91.659, 134.432, -160.954, 43.424, 166.352]
  MoveL 2871 to (-318.57, 36.27, -6.25) mm, rotated rx -179.9 ry 0 rz -90 deg; joints [12.98, -91.657, 134.432, -160.938, 43.429, 166.34]
  MoveL 2872 to (-316.39, 36.2, -6.26) mm, rotated rx -179.9 ry 0 rz -90 deg; joints [13.098, -91.619, 134.401, -160.773, 43.464, 166.224]
  MoveL 2873 to (-314.35, 36.12, -7.04) mm, rotated rx -179.9 ry 0 rz -90 deg; joints [13.199, -91.531, 134.323, -160.634, 43.498, 166.127]
  MoveL 2874 to (-312.72, 36.04, -8.51) mm, rotated rx -179.9 ry 0 rz -90 deg; joints [13.268, -91.404, 134.207, -160.541, 43.526, 166.063]
  MoveL 2875 to (-311.73, 35.97, -10.45) mm, rotated rx -179.9 ry 0 rz -90 deg; joints [13.297, -91.254, 134.07, -160.504, 43.545, 166.04]
  MoveL 2876 to (-311.49, 35.89, -12.63) mm, rotated rx -179.9 ry 0 rz -90 deg; joints [13.282, -91.101, 133.93, -160.53, 43.553, 166.062]
  MoveL 2877 to (-312.04, 35.81, -14.74) mm, rotated rx -179.9 ry 0 rz -90 deg; joints [13.225, -90.964, 133.806, -160.614, 43.551, 166.125]
  MoveL 2878 to (-313.31, 35.74, -16.52) mm, rotated rx -179.9 ry 0 rz -90 deg; joints [13.135, -90.861, 133.714, -160.746, 43.539, 166.221]
  MoveL 2879 to (-315.13, 35.66, -17.73) mm, rotated rx -179.9 ry 0 rz -90 deg; joints [13.021, -90.805, 133.667, -160.909, 43.521, 166.339]
  MoveL 2880 to (-317.26, 35.58, -18.21) mm, rotated rx -179.9 ry 0 rz -90 deg; joints [12.901, -90.802, 133.671, -161.082, 43.499, 166.465]
  MoveL 2881 to (-319.43, 35.51, -17.9) mm, rotated rx -179.9 ry 0 rz -90 deg; joints [12.788, -90.852, 133.727, -161.243, 43.478, 166.581]
  MoveL 2882 to (-321.34, 35.43, -16.84) mm, rotated rx -179.9 ry 0 rz -90 deg; joints [12.698, -90.949, 133.827, -161.371, 43.46, 166.673]
  MoveL 2883 to (-322.75, 35.35, -15.17) mm, rotated rx -179.9 ry 0 rz -90 deg; joints [12.643, -91.079, 133.959, -161.45, 43.449, 166.73]
  MoveL 2884 to (-323.47, 35.28, -13.1) mm, rotated rx -179.9 ry 0 rz -90 deg; joints [12.629, -91.225, 134.106, -161.469, 43.446, 166.744]
  MoveL 2885 to (-323.4, 35.2, -10.92) mm, rotated rx -179.9 ry 0 rz -90 deg; joints [12.659, -91.368, 134.248, -161.426, 43.452, 166.713]
  MoveL 2886 to (-322.56, 35.12, -8.9) mm, rotated rx -179.9 ry 0 rz -90 deg; joints [12.73, -91.489, 134.369, -161.327, 43.469, 166.642]
  MoveL 2887 to (-321.06, 35.05, -7.31) mm, rotated rx -179.9 ry 0 rz -90 deg; joints [12.831, -91.57, 134.451, -161.184, 43.494, 166.54]
  MoveL 2888 to (-319.09, 34.97, -6.36) mm, rotated rx -179.9 ry 0 rz -90 deg; joints [12.951, -91.601, 134.485, -161.017, 43.525, 166.421]
  MoveL 2889 to (-316.91, 34.89, -6.18) mm, rotated rx -179.9 ry 0 rz -90 deg; joints [13.071, -91.576, 134.467, -160.848, 43.56, 166.303]
  MoveL 2890 to (-314.81, 34.82, -6.79) mm, rotated rx -179.9 ry 0 rz -90 deg; joints [13.178, -91.499, 134.399, -160.702, 43.594, 166.2]
  MoveL 2891 to (-313.06, 34.74, -8.1) mm, rotated rx -179.9 ry 0 rz -90 deg; joints [13.256, -91.38, 134.291, -160.596, 43.623, 166.128]
  MoveL 2892 to (-311.9, 34.66, -9.95) mm, rotated rx -179.9 ry 0 rz -90 deg; joints [13.295, -91.234, 134.157, -160.545, 43.645, 166.094]
  MoveL 2893 to (-311.47, 34.59, -12.1) mm, rotated rx -179.9 ry 0 rz -90 deg; joints [13.29, -91.08, 134.016, -160.556, 43.656, 166.105]
  MoveL 2894 to (-311.84, 34.51, -14.25) mm, rotated rx -179.9 ry 0 rz -90 deg; joints [13.243, -90.938, 133.886, -160.627, 43.656, 166.158]
  MoveL 2895 to (-312.95, 34.43, -16.14) mm, rotated rx -179.9 ry 0 rz -90 deg; joints [13.16, -90.825, 133.785, -160.748, 43.646, 166.247]
  MoveL 2896 to (-314.65, 34.36, -17.5) mm, rotated rx -179.9 ry 0 rz -90 deg; joints [13.051, -90.757, 133.726, -160.905, 43.629, 166.361]
  MoveL 2897 to (-316.74, 34.28, -18.17) mm, rotated rx -179.9 ry 0 rz -90 deg; joints [12.93, -90.741, 133.718, -161.077, 43.608, 166.486]
  MoveL 2898 to (-318.92, 34.2, -18.05) mm, rotated rx -179.9 ry 0 rz -90 deg; joints [12.814, -90.778, 133.762, -161.242, 43.587, 166.605]
  MoveL 2899 to (-320.92, 34.13, -17.16) mm, rotated rx -179.9 ry 0 rz -90 deg; joints [12.718, -90.865, 133.852, -161.38, 43.568, 166.704]
  MoveL 2900 to (-322.47, 34.05, -15.62) mm, rotated rx -179.9 ry 0 rz -90 deg; joints [12.653, -90.988, 133.978, -161.472, 43.555, 166.77]
  MoveL 2901 to (-323.36, 33.97, -13.62) mm, rotated rx -179.9 ry 0 rz -90 deg; joints [12.629, -91.132, 134.123, -161.506, 43.55, 166.795]
  MoveL 2902 to (-323.49, 33.9, -11.44) mm, rotated rx -179.9 ry 0 rz -90 deg; joints [12.649, -91.278, 134.268, -161.478, 43.554, 166.775]
  MoveL 2903 to (-322.83, 33.82, -9.36) mm, rotated rx -179.9 ry 0 rz -90 deg; joints [12.71, -91.405, 134.395, -161.392, 43.568, 166.713]
  MoveL 2904 to (-321.47, 33.74, -7.64) mm, rotated rx -179.9 ry 0 rz -90 deg; joints [12.805, -91.497, 134.488, -161.258, 43.591, 166.617]
  MoveL 2905 to (-319.59, 33.66, -6.53) mm, rotated rx -179.9 ry 0 rz -90 deg; joints [12.922, -91.541, 134.534, -161.095, 43.622, 166.502]
  MoveL 2906 to (-317.44, 33.59, -6.15) mm, rotated rx -179.9 ry 0 rz -90 deg; joints [13.043, -91.53, 134.529, -160.925, 43.656, 166.382]
  MoveL 2907 to (-315.29, 33.51, -6.57) mm, rotated rx -179.9 ry 0 rz -90 deg; joints [13.155, -91.465, 134.472, -160.771, 43.69, 166.275]
  MoveL 2908 to (-313.44, 33.43, -7.73) mm, rotated rx -179.9 ry 0 rz -90 deg; joints [13.241, -91.355, 134.372, -160.654, 43.721, 166.194]
  MoveL 2909 to (-312.12, 33.36, -9.47) mm, rotated rx -179.9 ry 0 rz -90 deg; joints [13.29, -91.213, 134.243, -160.59, 43.744, 166.151]
  MoveL 2910 to (-311.5, 33.28, -11.57) mm, rotated rx -179.9 ry 0 rz -90 deg; joints [13.296, -91.059, 134.102, -160.585, 43.758, 166.151]
  MoveL 2911 to (-311.68, 33.2, -13.75) mm, rotated rx -179.9 ry 0 rz -90 deg; joints [13.259, -90.913, 133.968, -160.642, 43.76, 166.194]
  MoveL 2912 to (-312.62, 33.13, -15.72) mm, rotated rx -179.9 ry 0 rz -90 deg; joints [13.183, -90.792, 133.858, -160.752, 43.753, 166.275]
  MoveL 2913 to (-314.2, 33.05, -17.23) mm, rotated rx -179.9 ry 0 rz -90 deg; joints [13.079, -90.712, 133.788, -160.902, 43.737, 166.384]
  MoveL 2914 to (-316.21, 32.97, -18.08) mm, rotated rx -179.9 ry 0 rz -90 deg; joints [12.96, -90.683, 133.768, -161.072, 43.717, 166.506]
  MoveL 2915 to (-318.4, 32.9, -18.15) mm, rotated rx -179.9 ry 0 rz -90 deg; joints [12.842, -90.708, 133.799, -161.24, 43.696, 166.628]
  MoveL 2916 to (-320.47, 32.82, -17.44) mm, rotated rx -179.9 ry 0 rz -90 deg; joints [12.739, -90.783, 133.879, -161.386, 43.676, 166.733]
  MoveL 2917 to (-322.14, 32.74, -16.04) mm, rotated rx -179.9 ry 0 rz -90 deg; joints [12.666, -90.899, 133.998, -161.491, 43.662, 166.808]
  MoveL 2918 to (-323.21, 32.67, -14.13) mm, rotated rx -179.9 ry 0 rz -90 deg; joints [12.631, -91.039, 134.14, -161.54, 43.655, 166.843]
  MoveL 2919 to (-323.53, 32.59, -11.97) mm, rotated rx -179.9 ry 0 rz -90 deg; joints [12.64, -91.186, 134.287, -161.527, 43.657, 166.834]
  MoveL 2920 to (-323.06, 32.51, -9.83) mm, rotated rx -179.9 ry 0 rz -90 deg; joints [12.692, -91.32, 134.42, -161.453, 43.669, 166.781]
  MoveL 2921 to (-321.86, 32.44, -8.01) mm, rotated rx -179.9 ry 0 rz -90 deg; joints [12.78, -91.422, 134.522, -161.33, 43.69, 166.693]
  MoveL 2922 to (-320.08, 32.36, -6.73) mm, rotated rx -179.9 ry 0 rz -90 deg; joints [12.893, -91.478, 134.581, -161.172, 43.718, 166.582]
  MoveL 2923 to (-317.97, 32.28, -6.17) mm, rotated rx -179.9 ry 0 rz -90 deg; joints [13.015, -91.48, 134.588, -161.002, 43.752, 166.462]
  MoveL 2924 to (-315.79, 32.21, -6.4) mm, rotated rx -179.9 ry 0 rz -90 deg; joints [13.13, -91.427, 134.543, -160.843, 43.787, 166.351]
  MoveL 2925 to (-313.85, 32.13, -7.39) mm, rotated rx -179.9 ry 0 rz -90 deg; joints [13.224, -91.327, 134.452, -160.716, 43.818, 166.263]
  MoveL 2926 to (-312.38, 32.05, -9.01) mm, rotated rx -179.9 ry 0 rz -90 deg; joints [13.282, -91.192, 134.329, -160.637, 43.844, 166.21]
  MoveL 2927 to (-311.58, 31.98, -11.04) mm, rotated rx -179.9 ry 0 rz -90 deg; joints [13.299, -91.039, 134.189, -160.618, 43.859, 166.199]
  MoveL 2928 to (-311.56, 31.9, -13.23) mm, rotated rx -179.9 ry 0 rz -90 deg; joints [13.272, -90.889, 134.051, -160.66, 43.864, 166.232]
  MoveL 2929 to (-312.33, 31.82, -15.28) mm, rotated rx -179.9 ry 0 rz -90 deg; joints [13.205, -90.76, 133.934, -160.758, 43.859, 166.304]
  MoveL 2930 to (-313.77, 31.75, -16.92) mm, rotated rx -179.9 ry 0 rz -90 deg; joints [13.107, -90.67, 133.853, -160.9, 43.845, 166.407]
  MoveL 2931 to (-315.7, 31.67, -17.94) mm, rotated rx -179.9 ry 0 rz -90 deg; joints [12.99, -90.628, 133.82, -161.066, 43.826, 166.527]
  MoveL 2932 to (-317.87, 31.59, -18.21) mm, rotated rx -179.9 ry 0 rz -90 deg; joints [12.87, -90.639, 133.839, -161.237, 43.804, 166.65]
  MoveL 2933 to (-319.99, 31.52, -17.68) mm, rotated rx -179.9 ry 0 rz -90 deg; joints [12.762, -90.703, 133.908, -161.39, 43.784, 166.76]
  MoveL 2934 to (-321.79, 31.44, -16.43) mm, rotated rx -179.9 ry 0 rz -90 deg; joints [12.681, -90.81, 134.019, -161.506, 43.769, 166.843]
  MoveL 2935 to (-323.02, 31.36, -14.62) mm, rotated rx -179.9 ry 0 rz -90 deg; joints [12.636, -90.947, 134.157, -161.569, 43.76, 166.888]
  MoveL 2936 to (-323.53, 31.28, -12.5) mm, rotated rx -179.9 ry 0 rz -90 deg; joints [12.635, -91.094, 134.304, -161.571, 43.76, 166.89]
  MoveL 2937 to (-323.24, 31.21, -10.33) mm, rotated rx -179.9 ry 0 rz -90 deg; joints [12.677, -91.232, 134.443, -161.512, 43.77, 166.848]
  MoveL 2938 to (-322.21, 31.13, -8.41) mm, rotated rx -179.9 ry 0 rz -90 deg; joints [12.757, -91.343, 134.554, -161.399, 43.789, 166.768]
  MoveL 2939 to (-320.55, 31.05, -6.98) mm, rotated rx -179.9 ry 0 rz -90 deg; joints [12.865, -91.411, 134.624, -161.248, 43.816, 166.661]
  MoveL 2940 to (-318.5, 30.98, -6.23) mm, rotated rx -179.9 ry 0 rz -90 deg; joints [12.986, -91.426, 134.643, -161.08, 43.848, 166.542]
  MoveL 2941 to (-316.31, 30.9, -6.27) mm, rotated rx -179.9 ry 0 rz -90 deg; joints [13.104, -91.387, 134.611, -160.916, 43.883, 166.428]
  MoveL 2942 to (-314.28, 30.82, -7.09) mm, rotated rx -179.9 ry 0 rz -90 deg; joints [13.204, -91.297, 134.53, -160.78, 43.916, 166.333]
  MoveL 2943 to (-312.67, 30.75, -8.57) mm, rotated rx -179.9 ry 0 rz -90 deg; joints [13.272, -91.169, 134.413, -160.688, 43.943, 166.271]
  MoveL 2944 to (-311.7, 30.67, -10.53) mm, rotated rx -179.9 ry 0 rz -90 deg; joints [13.3, -91.019, 134.275, -160.654, 43.961, 166.25]
  MoveL 2945 to (-311.49, 30.59, -12.7) mm, rotated rx -179.9 ry 0 rz -90 deg; joints [13.283, -90.866, 134.135, -160.681, 43.968, 166.272]
  MoveL 2946 to (-312.07, 30.52, -14.81) mm, rotated rx -179.9 ry 0 rz -90 deg; joints [13.225, -90.731, 134.011, -160.767, 43.965, 166.335]
  MoveL 2947 to (-313.37, 30.44, -16.58) mm, rotated rx -179.9 ry 0 rz -90 deg; joints [13.133, -90.63, 133.921, -160.899, 43.953, 166.431]
  MoveL 2948 to (-315.2, 30.36, -17.76) mm, rotated rx -179.9 ry 0 rz -90 deg; joints [13.019, -90.575, 133.875, -161.061, 43.935, 166.548]
  MoveL 2949 to (-317.34, 30.29, -18.21) mm, rotated rx -179.9 ry 0 rz -90 deg; joints [12.899, -90.574, 133.882, -161.233, 43.914, 166.671]
  MoveL 2950 to (-319.5, 30.21, -17.88) mm, rotated rx -179.9 ry 0 rz -90 deg; joints [12.787, -90.626, 133.939, -161.392, 43.893, 166.786]
  MoveL 2951 to (-321.4, 30.13, -16.79) mm, rotated rx -179.9 ry 0 rz -90 deg; joints [12.698, -90.724, 134.041, -161.518, 43.876, 166.876]
  MoveL 2952 to (-322.79, 30.06, -15.1) mm, rotated rx -179.9 ry 0 rz -90 deg; joints [12.644, -90.854, 134.174, -161.595, 43.866, 166.931]
  MoveL 2953 to (-323.48, 29.98, -13.03) mm, rotated rx -179.9 ry 0 rz -90 deg; joints [12.631, -91, 134.321, -161.612, 43.864, 166.943]
  MoveL 2954 to (-323.38, 29.9, -10.84) mm, rotated rx -179.9 ry 0 rz -90 deg; joints [12.663, -91.143, 134.464, -161.567, 43.871, 166.912]
  MoveL 2955 to (-322.52, 29.83, -8.83) mm, rotated rx -179.9 ry 0 rz -90 deg; joints [12.735, -91.262, 134.583, -161.467, 43.888, 166.84]
  MoveL 2956 to (-321, 29.75, -7.27) mm, rotated rx -179.9 ry 0 rz -90 deg; joints [12.838, -91.341, 134.664, -161.323, 43.913, 166.739]
  MoveL 2957 to (-319.01, 29.67, -6.34) mm, rotated rx -179.9 ry 0 rz -90 deg; joints [12.957, -91.37, 134.696, -161.157, 43.945, 166.622]
  MoveL 2958 to (-316.83, 29.6, -6.19) mm, rotated rx -179.9 ry 0 rz -90 deg; joints [13.078, -91.343, 134.676, -160.991, 43.979, 166.506]
  MoveL 2959 to (-314.74, 29.52, -6.82) mm, rotated rx -179.9 ry 0 rz -90 deg; joints [13.183, -91.265, 134.606, -160.846, 44.013, 166.405]
  MoveL 2960 to (-313.01, 29.44, -8.16) mm, rotated rx -179.9 ry 0 rz -90 deg; joints [13.26, -91.145, 134.497, -160.742, 44.041, 166.334]
  MoveL 2961 to (-311.87, 29.37, -10.03) mm, rotated rx -179.9 ry 0 rz -90 deg; joints [13.298, -90.998, 134.362, -160.694, 44.061, 166.303]
  MoveL 2962 to (-311.47, 29.29, -12.17) mm, rotated rx -179.9 ry 0 rz -90 deg; joints [13.292, -90.845, 134.22, -160.706, 44.071, 166.314]
  MoveL 2963 to (-311.86, 29.21, -14.33) mm, rotated rx -179.9 ry 0 rz -90 deg; joints [13.243, -90.703, 134.091, -160.778, 44.071, 166.368]
  MoveL 2964 to (-313, 29.14, -16.19) mm, rotated rx -179.9 ry 0 rz -90 deg; joints [13.158, -90.593, 133.991, -160.9, 44.06, 166.457]
  MoveL 2965 to (-314.72, 29.06, -17.54) mm, rotated rx -179.9 ry 0 rz -90 deg; joints [13.049, -90.526, 133.934, -161.056, 44.043, 166.569]
  MoveL 2966 to (-316.81, 28.98, -18.18) mm, rotated rx -179.9 ry 0 rz -90 deg; joints [12.928, -90.512, 133.927, -161.228, 44.023, 166.692]
  MoveL 2967 to (-318.99, 28.9, -18.03) mm, rotated rx -179.9 ry 0 rz -90 deg; joints [12.813, -90.551, 133.973, -161.391, 44.002, 166.81]
  MoveL 2968 to (-320.98, 28.83, -17.11) mm, rotated rx -179.9 ry 0 rz -90 deg; joints [12.717, -90.639, 134.065, -161.527, 43.984, 166.907]
  MoveL 2969 to (-322.51, 28.75, -15.55) mm, rotated rx -179.9 ry 0 rz -90 deg; joints [12.653, -90.763, 134.192, -161.617, 43.972, 166.971]
  MoveL 2970 to (-323.38, 28.67, -13.55) mm, rotated rx -179.9 ry 0 rz -90 deg; joints [12.631, -90.907, 134.338, -161.649, 43.968, 166.994]
  MoveL 2971 to (-323.48, 28.6, -11.36) mm, rotated rx -179.9 ry 0 rz -90 deg; joints [12.652, -91.052, 134.483, -161.619, 43.974, 166.973]
  MoveL 2972 to (-322.79, 28.52, -9.29) mm, rotated rx -179.9 ry 0 rz -90 deg; joints [12.715, -91.178, 134.609, -161.531, 43.988, 166.911]
  MoveL 2973 to (-321.41, 28.44, -7.59) mm, rotated rx -179.9 ry 0 rz -90 deg; joints [12.811, -91.268, 134.701, -161.397, 44.012, 166.816]
  MoveL 2974 to (-319.52, 28.37, -6.5) mm, rotated rx -179.9 ry 0 rz -90 deg; joints [12.928, -91.31, 134.745, -161.234, 44.042, 166.702]
  MoveL 2975 to (-317.36, 28.29, -6.15) mm, rotated rx -179.9 ry 0 rz -90 deg; joints [13.05, -91.296, 134.738, -161.066, 44.076, 166.584]
  MoveL 2976 to (-315.22, 28.21, -6.6) mm, rotated rx -179.9 ry 0 rz -90 deg; joints [13.16, -91.23, 134.679, -160.914, 44.11, 166.479]
  MoveL 2977 to (-313.38, 28.14, -7.78) mm, rotated rx -179.9 ry 0 rz -90 deg; joints [13.245, -91.118, 134.578, -160.799, 44.139, 166.4]
  MoveL 2978 to (-312.08, 28.06, -9.54) mm, rotated rx -179.9 ry 0 rz -90 deg; joints [13.293, -90.977, 134.448, -160.737, 44.161, 166.358]
  MoveL 2979 to (-311.5, 27.98, -11.65) mm, rotated rx -179.9 ry 0 rz -90 deg; joints [13.298, -90.823, 134.306, -160.734, 44.174, 166.359]
  MoveL 2980 to (-311.7, 27.91, -13.82) mm, rotated rx -179.9 ry 0 rz -90 deg; joints [13.259, -90.677, 134.172, -160.792, 44.176, 166.403]
  MoveL 2981 to (-312.66, 27.83, -15.78) mm, rotated rx -179.9 ry 0 rz -90 deg; joints [13.182, -90.558, 134.063, -160.903, 44.168, 166.484]
  MoveL 2982 to (-314.26, 27.75, -17.27) mm, rotated rx -179.9 ry 0 rz -90 deg; joints [13.077, -90.48, 133.995, -161.053, 44.152, 166.592]
  MoveL 2983 to (-316.29, 27.68, -18.09) mm, rotated rx -179.9 ry 0 rz -90 deg; joints [12.958, -90.452, 133.976, -161.222, 44.132, 166.713]
  MoveL 2984 to (-318.48, 27.6, -18.14) mm, rotated rx -179.9 ry 0 rz -90 deg; joints [12.84, -90.479, 134.009, -161.389, 44.111, 166.833]
  MoveL 2985 to (-320.53, 27.52, -17.4) mm, rotated rx -179.9 ry 0 rz -90 deg; joints [12.738, -90.556, 134.091, -161.533, 44.092, 166.935]
  MoveL 2986 to (-322.19, 27.45, -15.98) mm, rotated rx -179.9 ry 0 rz -90 deg; joints [12.666, -90.672, 134.211, -161.635, 44.079, 167.008]
  MoveL 2987 to (-323.24, 27.37, -14.06) mm, rotated rx -179.9 ry 0 rz -90 deg; joints [12.633, -90.813, 134.354, -161.682, 44.073, 167.042]
  MoveL 2988 to (-323.53, 27.29, -11.89) mm, rotated rx -179.9 ry 0 rz -90 deg; joints [12.644, -90.96, 134.501, -161.667, 44.076, 167.031]
  MoveL 2989 to (-323.03, 27.22, -9.76) mm, rotated rx -179.9 ry 0 rz -90 deg; joints [12.697, -91.092, 134.634, -161.592, 44.089, 166.979]
  MoveL 2990 to (-321.8, 27.14, -7.95) mm, rotated rx -179.9 ry 0 rz -90 deg; joints [12.786, -91.192, 134.735, -161.468, 44.11, 166.891]
  MoveL 2991 to (-320.01, 27.06, -6.7) mm, rotated rx -179.9 ry 0 rz -90 deg; joints [12.899, -91.246, 134.792, -161.311, 44.139, 166.781]
  MoveL 2992 to (-317.89, 26.99, -6.16) mm, rotated rx -179.9 ry 0 rz -90 deg; joints [13.021, -91.246, 134.797, -161.142, 44.172, 166.663]
  MoveL 2993 to (-315.72, 26.91, -6.42) mm, rotated rx -179.9 ry 0 rz -90 deg; joints [13.136, -91.192, 134.75, -160.985, 44.206, 166.553]
  MoveL 2994 to (-313.78, 26.83, -7.44) mm, rotated rx -179.9 ry 0 rz -90 deg; joints [13.228, -91.09, 134.658, -160.859, 44.237, 166.467]
  MoveL 2995 to (-312.34, 26.76, -9.07) mm, rotated rx -179.9 ry 0 rz -90 deg; joints [13.286, -90.954, 134.533, -160.783, 44.261, 166.416]
  MoveL 2996 to (-311.57, 26.68, -11.12) mm, rotated rx -179.9 ry 0 rz -90 deg; joints [13.301, -90.802, 134.392, -160.766, 44.276, 166.407]
  MoveL 2997 to (-311.58, 26.6, -13.31) mm, rotated rx -179.9 ry 0 rz -90 deg; joints [13.273, -90.652, 134.255, -160.81, 44.28, 166.44]
  MoveL 2998 to (-312.37, 26.53, -15.34) mm, rotated rx -179.9 ry 0 rz -90 deg; joints [13.204, -90.525, 134.138, -160.908, 44.274, 166.512]
  MoveL 2999 to (-313.83, 26.45, -16.97) mm, rotated rx -179.9 ry 0 rz -90 deg; joints [13.105, -90.436, 134.059, -161.05, 44.26, 166.614]
  MoveL 3000 to (-315.78, 26.37, -17.96) mm, rotated rx -179.9 ry 0 rz -90 deg; joints [12.988, -90.396, 134.027, -161.216, 44.241, 166.733]
  MoveL 3001 to (-317.95, 26.29, -18.2) mm, rotated rx -179.9 ry 0 rz -90 deg; joints [12.868, -90.41, 134.048, -161.386, 44.22, 166.854]
  MoveL 3002 to (-320.06, 26.22, -17.65) mm, rotated rx -179.9 ry 0 rz -90 deg; joints [12.761, -90.475, 134.119, -161.537, 44.201, 166.962]
  MoveL 3003 to (-321.84, 26.14, -16.38) mm, rotated rx -179.9 ry 0 rz -90 deg; joints [12.68, -90.583, 134.231, -161.65, 44.186, 167.043]
  MoveL 3004 to (-323.05, 26.06, -14.55) mm, rotated rx -179.9 ry 0 rz -90 deg; joints [12.637, -90.719, 134.37, -161.711, 44.179, 167.087]
  MoveL 3005 to (-323.53, 25.99, -12.42) mm, rotated rx -179.9 ry 0 rz -90 deg; joints [12.638, -90.866, 134.518, -161.711, 44.18, 167.087]
  MoveL 3006 to (-323.22, 25.91, -10.26) mm, rotated rx -179.9 ry 0 rz -90 deg; joints [12.681, -91.004, 134.656, -161.651, 44.19, 167.045]
  MoveL 3007 to (-322.16, 25.83, -8.35) mm, rotated rx -179.9 ry 0 rz -90 deg; joints [12.762, -91.113, 134.766, -161.537, 44.21, 166.965]
  MoveL 3008 to (-320.48, 25.76, -6.94) mm, rotated rx -179.9 ry 0 rz -90 deg; joints [12.871, -91.179, 134.835, -161.386, 44.237, 166.859]
  MoveL 3009 to (-318.42, 25.68, -6.22) mm, rotated rx -179.9 ry 0 rz -90 deg; joints [12.993, -91.192, 134.852, -161.219, 44.269, 166.742]
  MoveL 3010 to (-316.23, 25.6, -6.29) mm, rotated rx -179.9 ry 0 rz -90 deg; joints [13.111, -91.151, 134.818, -161.057, 44.303, 166.629]
  MoveL 3011 to (-314.22, 25.53, -7.13) mm, rotated rx -179.9 ry 0 rz -90 deg; joints [13.209, -91.06, 134.736, -160.922, 44.335, 166.537]
  MoveL 3012 to (-312.63, 25.45, -8.63) mm, rotated rx -179.9 ry 0 rz -90 deg; joints [13.276, -90.931, 134.617, -160.833, 44.361, 166.476]
  MoveL 3013 to (-311.68, 25.37, -10.6) mm, rotated rx -179.9 ry 0 rz -90 deg; joints [13.302, -90.781, 134.479, -160.801, 44.378, 166.456]
  MoveL 3014 to (-311.5, 25.3, -12.78) mm, rotated rx -179.9 ry 0 rz -90 deg; joints [13.284, -90.629, 134.338, -160.83, 44.384, 166.48]
  MoveL 3015 to (-312.11, 25.22, -14.88) mm, rotated rx -179.9 ry 0 rz -90 deg; joints [13.224, -90.495, 134.215, -160.916, 44.381, 166.543]
  MoveL 3016 to (-313.42, 25.14, -16.63) mm, rotated rx -179.9 ry 0 rz -90 deg; joints [13.131, -90.395, 134.126, -161.049, 44.368, 166.638]
  MoveL 3017 to (-315.28, 25.07, -17.79) mm, rotated rx -179.9 ry 0 rz -90 deg; joints [13.017, -90.342, 134.082, -161.21, 44.35, 166.754]
  MoveL 3018 to (-317.42, 24.99, -18.22) mm, rotated rx -179.9 ry 0 rz -90 deg; joints [12.897, -90.343, 134.09, -161.381, 44.329, 166.876]
  MoveL 3019 to (-319.57, 24.91, -17.85) mm, rotated rx -179.9 ry 0 rz -90 deg; joints [12.785, -90.396, 134.149, -161.538, 44.309, 166.988]
  MoveL 3020 to (-321.46, 24.84, -16.74) mm, rotated rx -179.9 ry 0 rz -90 deg; joints [12.697, -90.495, 134.253, -161.662, 44.294, 167.076]
  MoveL 3021 to (-322.82, 24.76, -15.03) mm, rotated rx -179.9 ry 0 rz -90 deg; joints [12.644, -90.626, 134.387, -161.737, 44.284, 167.129]
  MoveL 3022 to (-323.49, 24.68, -12.95) mm, rotated rx -179.9 ry 0 rz -90 deg; joints [12.634, -90.772, 134.534, -161.752, 44.283, 167.14]
  MoveL 3023 to (-323.37, 24.61, -10.77) mm, rotated rx -179.9 ry 0 rz -90 deg; joints [12.667, -90.914, 134.677, -161.705, 44.292, 167.108]
  MoveL 3024 to (-322.48, 24.53, -8.77) mm, rotated rx -179.9 ry 0 rz -90 deg; joints [12.74, -91.031, 134.795, -161.604, 44.309, 167.037]
  MoveL 3025 to (-320.93, 24.45, -7.22) mm, rotated rx -179.9 ry 0 rz -90 deg; joints [12.844, -91.109, 134.875, -161.461, 44.335, 166.936]
  MoveL 3026 to (-318.94, 24.38, -6.33) mm, rotated rx -179.9 ry 0 rz -90 deg; joints [12.963, -91.135, 134.905, -161.295, 44.366, 166.821]
  MoveL 3027 to (-316.76, 24.3, -6.2) mm, rotated rx -179.9 ry 0 rz -90 deg; joints [13.084, -91.107, 134.883, -161.13, 44.4, 166.706]
  MoveL 3028 to (-314.67, 24.22, -6.86) mm, rotated rx -179.9 ry 0 rz -90 deg; joints [13.189, -91.027, 134.811, -160.987, 44.433, 166.607]
  MoveL 3029 to (-312.96, 24.15, -8.22) mm, rotated rx -179.9 ry 0 rz -90 deg; joints [13.264, -90.906, 134.7, -160.886, 44.46, 166.539]
  MoveL 3030 to (-311.84, 24.07, -10.1) mm, rotated rx -179.9 ry 0 rz -90 deg; joints [13.3, -90.759, 134.565, -160.839, 44.479, 166.509]
  MoveL 3031 to (-311.47, 23.99, -12.25) mm, rotated rx -179.9 ry 0 rz -90 deg; joints [13.293, -90.606, 134.423, -160.854, 44.488, 166.521]
  MoveL 3032 to (-311.89, 23.92, -14.4) mm, rotated rx -179.9 ry 0 rz -90 deg; joints [13.243, -90.466, 134.294, -160.927, 44.487, 166.575]
  MoveL 3033 to (-313.05, 23.84, -16.25) mm, rotated rx -179.9 ry 0 rz -90 deg; joints [13.157, -90.357, 134.195, -161.049, 44.476, 166.664]
  MoveL 3034 to (-314.79, 23.76, -17.57) mm, rotated rx -179.9 ry 0 rz -90 deg; joints [13.047, -90.292, 134.139, -161.205, 44.459, 166.775]
  MoveL 3035 to (-316.89, 23.68, -18.19) mm, rotated rx -179.9 ry 0 rz -90 deg; joints [12.926, -90.279, 134.135, -161.375, 44.439, 166.896]
  MoveL 3036 to (-319.07, 23.61, -18.01) mm, rotated rx -179.9 ry 0 rz -90 deg; joints [12.811, -90.32, 134.182, -161.537, 44.418, 167.012]
  MoveL 3037 to (-321.04, 23.53, -17.07) mm, rotated rx -179.9 ry 0 rz -90 deg; joints [12.716, -90.409, 134.276, -161.671, 44.402, 167.107]
  MoveL 3038 to (-322.55, 23.45, -15.49) mm, rotated rx -179.9 ry 0 rz -90 deg; joints [12.654, -90.534, 134.404, -161.758, 44.391, 167.169]
  MoveL 3039 to (-323.4, 23.38, -13.47) mm, rotated rx -179.9 ry 0 rz -90 deg; joints [12.633, -90.678, 134.55, -161.788, 44.388, 167.19]
  MoveL 3040 to (-323.47, 23.3, -11.29) mm, rotated rx -179.9 ry 0 rz -90 deg; joints [12.656, -90.822, 134.695, -161.757, 44.394, 167.169]
  MoveL 3041 to (-322.76, 23.22, -9.22) mm, rotated rx -179.9 ry 0 rz -90 deg; joints [12.72, -90.947, 134.821, -161.668, 44.41, 167.106]
  MoveL 3042 to (-321.36, 23.15, -7.54) mm, rotated rx -179.9 ry 0 rz -90 deg; joints [12.817, -91.035, 134.911, -161.533, 44.433, 167.012]
  MoveL 3043 to (-319.45, 23.07, -6.47) mm, rotated rx -179.9 ry 0 rz -90 deg; joints [12.934, -91.075, 134.954, -161.371, 44.464, 166.899]
  MoveL 3044 to (-317.28, 22.99, -6.16) mm, rotated rx -179.9 ry 0 rz -90 deg; joints [13.056, -91.06, 134.945, -161.204, 44.497, 166.783]
  MoveL 3045 to (-315.15, 22.92, -6.63) mm, rotated rx -179.9 ry 0 rz -90 deg; joints [13.166, -90.991, 134.884, -161.054, 44.53, 166.68]
  MoveL 3046 to (-313.33, 22.84, -7.83) mm, rotated rx -179.9 ry 0 rz -90 deg; joints [13.25, -90.879, 134.782, -160.942, 44.559, 166.603]
  MoveL 3047 to (-312.05, 22.76, -9.61) mm, rotated rx -179.9 ry 0 rz -90 deg; joints [13.296, -90.737, 134.65, -160.881, 44.58, 166.563]
  MoveL 3048 to (-311.49, 22.69, -11.72) mm, rotated rx -179.9 ry 0 rz -90 deg; joints [13.299, -90.583, 134.508, -160.881, 44.591, 166.565]
  MoveL 3049 to (-311.72, 22.61, -13.9) mm, rotated rx -179.9 ry 0 rz -90 deg; joints [13.259, -90.438, 134.374, -160.94, 44.592, 166.61]
  MoveL 3050 to (-312.71, 22.53, -15.85) mm, rotated rx -179.9 ry 0 rz -90 deg; joints [13.181, -90.32, 134.266, -161.051, 44.584, 166.69]
  MoveL 3051 to (-314.33, 22.46, -17.31) mm, rotated rx -179.9 ry 0 rz -90 deg; joints [13.075, -90.244, 134.199, -161.201, 44.568, 166.797]
  MoveL 3052 to (-316.37, 22.38, -18.11) mm, rotated rx -179.9 ry 0 rz -90 deg; joints [12.956, -90.219, 134.182, -161.369, 44.548, 166.917]
  MoveL 3053 to (-318.55, 22.3, -18.13) mm, rotated rx -179.9 ry 0 rz -90 deg; joints [12.838, -90.247, 134.217, -161.535, 44.527, 167.035]
  MoveL 3054 to (-320.6, 22.23, -17.36) mm, rotated rx -179.9 ry 0 rz -90 deg; joints [12.737, -90.325, 134.301, -161.677, 44.51, 167.135]
  MoveL 3055 to (-322.24, 22.15, -15.92) mm, rotated rx -179.9 ry 0 rz -90 deg; joints [12.666, -90.442, 134.422, -161.777, 44.498, 167.206]
  MoveL 3056 to (-323.26, 22.07, -13.98) mm, rotated rx -179.9 ry 0 rz -90 deg; joints [12.635, -90.583, 134.566, -161.821, 44.493, 167.238]
  MoveL 3057 to (-323.52, 22, -11.81) mm, rotated rx -179.9 ry 0 rz -90 deg; joints [12.647, -90.729, 134.713, -161.805, 44.497, 167.227]
  MoveL 3058 to (-323, 21.92, -9.69) mm, rotated rx -179.9 ry 0 rz -90 deg; joints [12.702, -90.86, 134.845, -161.729, 44.51, 167.174]
  MoveL 3059 to (-321.75, 21.84, -7.9) mm, rotated rx -179.9 ry 0 rz -90 deg; joints [12.792, -90.959, 134.945, -161.604, 44.532, 167.087]
  MoveL 3060 to (-319.94, 21.77, -6.67) mm, rotated rx -179.9 ry 0 rz -90 deg; joints [12.906, -91.011, 135, -161.447, 44.561, 166.977]
  MoveL 3061 to (-317.81, 21.69, -6.16) mm, rotated rx -179.9 ry 0 rz -90 deg; joints [13.028, -91.009, 135.004, -161.279, 44.594, 166.861]
  MoveL 3062 to (-315.65, 21.61, -6.44) mm, rotated rx -179.9 ry 0 rz -90 deg; joints [13.142, -90.953, 134.955, -161.123, 44.627, 166.754]
  MoveL 3063 to (-313.72, 21.54, -7.48) mm, rotated rx -179.9 ry 0 rz -90 deg; joints [13.233, -90.85, 134.861, -161, 44.657, 166.669]
  MoveL 3064 to (-312.3, 21.46, -9.14) mm, rotated rx -179.9 ry 0 rz -90 deg; joints [13.289, -90.714, 134.735, -160.926, 44.68, 166.62]
  MoveL 3065 to (-311.55, 21.38, -11.2) mm, rotated rx -179.9 ry 0 rz -90 deg; joints [13.303, -90.561, 134.594, -160.911, 44.694, 166.612]
  MoveL 3066 to (-311.59, 21.3, -13.38) mm, rotated rx -179.9 ry 0 rz -90 deg; joints [13.273, -90.413, 134.456, -160.956, 44.697, 166.646]
  MoveL 3067 to (-312.41, 21.23, -15.41) mm, rotated rx -179.9 ry 0 rz -90 deg; joints [13.203, -90.287, 134.34, -161.056, 44.691, 166.718]
  MoveL 3068 to (-313.89, 21.15, -17.02) mm, rotated rx -179.9 ry 0 rz -90 deg; joints [13.103, -90.199, 134.262, -161.198, 44.676, 166.819]
  MoveL 3069 to (-315.85, 21.07, -17.99) mm, rotated rx -179.9 ry 0 rz -90 deg; joints [12.985, -90.161, 134.233, -161.363, 44.657, 166.937]
  MoveL 3070 to (-318.03, 21, -18.19) mm, rotated rx -179.9 ry 0 rz -90 deg; joints [12.866, -90.176, 134.255, -161.531, 44.637, 167.056]
  MoveL 3071 to (-320.13, 20.92, -17.61) mm, rotated rx -179.9 ry 0 rz -90 deg; joints [12.759, -90.243, 134.328, -161.68, 44.618, 167.162]
  MoveL 3072 to (-321.9, 20.84, -16.32) mm, rotated rx -179.9 ry 0 rz -90 deg; joints [12.68, -90.352, 134.441, -161.792, 44.605, 167.241]
  MoveL 3073 to (-323.08, 20.77, -14.48) mm, rotated rx -179.9 ry 0 rz -90 deg; joints [12.639, -90.489, 134.581, -161.85, 44.598, 167.283]
  MoveL 3074 to (-323.53, 20.69, -12.34) mm, rotated rx -179.9 ry 0 rz -90 deg; joints [12.64, -90.635, 134.73, -161.848, 44.6, 167.282]
  MoveL 3075 to (-323.19, 20.61, -10.18) mm, rotated rx -179.9 ry 0 rz -90 deg; joints [12.685, -90.772, 134.867, -161.786, 44.612, 167.239]
  MoveL 3076 to (-322.11, 20.54, -8.29) mm, rotated rx -179.9 ry 0 rz -90 deg; joints [12.768, -90.879, 134.976, -161.672, 44.632, 167.159]
  MoveL 3077 to (-320.42, 20.46, -6.9) mm, rotated rx -179.9 ry 0 rz -90 deg; joints [12.877, -90.943, 135.043, -161.522, 44.659, 167.055]
  MoveL 3078 to (-318.34, 20.38, -6.21) mm, rotated rx -179.9 ry 0 rz -90 deg; joints [12.999, -90.955, 135.059, -161.355, 44.691, 166.939]
  MoveL 3079 to (-316.16, 20.31, -6.3) mm, rotated rx -179.9 ry 0 rz -90 deg; joints [13.117, -90.912, 135.023, -161.194, 44.725, 166.828]
  MoveL 3080 to (-314.15, 20.23, -7.17) mm, rotated rx -179.9 ry 0 rz -90 deg; joints [13.215, -90.819, 134.939, -161.062, 44.756, 166.738]
  MoveL 3081 to (-312.58, 20.15, -8.69) mm, rotated rx -179.9 ry 0 rz -90 deg; joints [13.28, -90.689, 134.819, -160.975, 44.781, 166.679]
  MoveL 3082 to (-311.66, 20.08, -10.68) mm, rotated rx -179.9 ry 0 rz -90 deg; joints [13.304, -90.539, 134.68, -160.945, 44.796, 166.661]
  MoveL 3083 to (-311.51, 20, -12.86) mm, rotated rx -179.9 ry 0 rz -90 deg; joints [13.285, -90.388, 134.539, -160.976, 44.802, 166.685]
  MoveL 3084 to (-312.14, 19.92, -14.95) mm, rotated rx -179.9 ry 0 rz -90 deg; joints [13.224, -90.255, 134.416, -161.063, 44.798, 166.748]
  MoveL 3085 to (-313.48, 19.85, -16.68) mm, rotated rx -179.9 ry 0 rz -90 deg; joints [13.13, -90.157, 134.328, -161.196, 44.785, 166.843]
  MoveL 3086 to (-315.35, 19.77, -17.82) mm, rotated rx -179.9 ry 0 rz -90 deg; joints [13.015, -90.106, 134.286, -161.357, 44.767, 166.958]
  MoveL 3087 to (-317.5, 19.69, -18.22) mm, rotated rx -179.9 ry 0 rz -90 deg; joints [12.895, -90.109, 134.296, -161.526, 44.746, 167.077]
  MoveL 3088 to (-319.65, 19.62, -17.82) mm, rotated rx -179.9 ry 0 rz -90 deg; joints [12.784, -90.164, 134.357, -161.681, 44.727, 167.187]
  MoveL 3089 to (-321.52, 19.54, -16.69) mm, rotated rx -179.9 ry 0 rz -90 deg; joints [12.697, -90.263, 134.462, -161.803, 44.712, 167.274]
  MoveL 3090 to (-322.86, 19.46, -14.96) mm, rotated rx -179.9 ry 0 rz -90 deg; joints [12.645, -90.395, 134.597, -161.876, 44.704, 167.325]
  MoveL 3091 to (-323.5, 19.39, -12.87) mm, rotated rx -179.9 ry 0 rz -90 deg; joints [12.637, -90.541, 134.745, -161.889, 44.704, 167.335]
  MoveL 3092 to (-323.35, 19.31, -10.69) mm, rotated rx -179.9 ry 0 rz -90 deg; joints [12.671, -90.681, 134.887, -161.841, 44.714, 167.302]
  MoveL 3093 to (-322.43, 19.23, -8.71) mm, rotated rx -179.9 ry 0 rz -90 deg; joints [12.746, -90.797, 135.005, -161.738, 44.732, 167.23]
  MoveL 3094 to (-320.87, 19.16, -7.18) mm, rotated rx -179.9 ry 0 rz -90 deg; joints [12.85, -90.873, 135.083, -161.595, 44.758, 167.131]
  MoveL 3095 to (-318.86, 19.08, -6.31) mm, rotated rx -179.9 ry 0 rz -90 deg; joints [12.97, -90.897, 135.112, -161.43, 44.789, 167.017]
  MoveL 3096 to (-316.68, 19, -6.21) mm, rotated rx -179.9 ry 0 rz -90 deg; joints [13.09, -90.867, 135.087, -161.267, 44.822, 166.904]
  MoveL 3097 to (-314.6, 18.92, -6.89) mm, rotated rx -179.9 ry 0 rz -90 deg; joints [13.194, -90.786, 135.014, -161.126, 44.854, 166.807]
  MoveL 3098 to (-312.91, 18.85, -8.28) mm, rotated rx -179.9 ry 0 rz -90 deg; joints [13.268, -90.663, 134.902, -161.026, 44.88, 166.741]
  MoveL 3099 to (-311.82, 18.77, -10.17) mm, rotated rx -179.9 ry 0 rz -90 deg; joints [13.303, -90.516, 134.765, -160.982, 44.898, 166.712]
  MoveL 3100 to (-311.47, 18.69, -12.33) mm, rotated rx -179.9 ry 0 rz -90 deg; joints [13.294, -90.364, 134.623, -160.998, 44.906, 166.726]
  MoveL 3101 to (-311.92, 18.62, -14.47) mm, rotated rx -179.9 ry 0 rz -90 deg; joints [13.242, -90.225, 134.494, -161.072, 44.904, 166.78]
  MoveL 3102 to (-313.1, 18.54, -16.31) mm, rotated rx -179.9 ry 0 rz -90 deg; joints [13.155, -90.117, 134.396, -161.195, 44.893, 166.868]
  MoveL 3103 to (-314.86, 18.46, -17.61) mm, rotated rx -179.9 ry 0 rz -90 deg; joints [13.044, -90.054, 134.342, -161.351, 44.876, 166.978]
  MoveL 3104 to (-316.97, 18.39, -18.19) mm, rotated rx -179.9 ry 0 rz -90 deg; joints [12.924, -90.044, 134.34, -161.52, 44.856, 167.098]
  MoveL 3105 to (-319.14, 18.31, -17.99) mm, rotated rx -179.9 ry 0 rz -90 deg; joints [12.809, -90.086, 134.389, -161.681, 44.836, 167.211]
  MoveL 3106 to (-321.11, 18.23, -17.02) mm, rotated rx -179.9 ry 0 rz -90 deg; joints [12.715, -90.176, 134.484, -161.812, 44.82, 167.304]
  MoveL 3107 to (-322.59, 18.16, -15.42) mm, rotated rx -179.9 ry 0 rz -90 deg; joints [12.655, -90.302, 134.614, -161.897, 44.811, 167.365]
  MoveL 3108 to (-323.41, 18.08, -13.4) mm, rotated rx -179.9 ry 0 rz -90 deg; joints [12.635, -90.446, 134.76, -161.925, 44.809, 167.385]
  MoveL 3109 to (-323.46, 18, -11.21) mm, rotated rx -179.9 ry 0 rz -90 deg; joints [12.66, -90.589, 134.906, -161.892, 44.816, 167.362]
  MoveL 3110 to (-322.72, 17.93, -9.15) mm, rotated rx -179.9 ry 0 rz -90 deg; joints [12.725, -90.712, 135.031, -161.802, 44.832, 167.299]
  MoveL 3111 to (-321.3, 17.85, -7.49) mm, rotated rx -179.9 ry 0 rz -90 deg; joints [12.823, -90.799, 135.12, -161.667, 44.857, 167.206]
  MoveL 3112 to (-319.37, 17.77, -6.45) mm, rotated rx -179.9 ry 0 rz -90 deg; joints [12.941, -90.836, 135.161, -161.506, 44.887, 167.094]
  MoveL 3113 to (-317.21, 17.7, -6.16) mm, rotated rx -179.9 ry 0 rz -90 deg; joints [13.062, -90.819, 135.149, -161.34, 44.92, 166.98]
  MoveL 3114 to (-315.08, 17.62, -6.66) mm, rotated rx -179.9 ry 0 rz -90 deg; joints [13.172, -90.749, 135.087, -161.192, 44.952, 166.879]
  MoveL 3115 to (-313.27, 17.54, -7.89) mm, rotated rx -179.9 ry 0 rz -90 deg; joints [13.254, -90.636, 134.983, -161.081, 44.98, 166.804]
  MoveL 3116 to (-312.02, 17.47, -9.68) mm, rotated rx -179.9 ry 0 rz -90 deg; joints [13.299, -90.493, 134.85, -161.023, 45, 166.766]
  MoveL 3117 to (-311.48, 17.39, -11.8) mm, rotated rx -179.9 ry 0 rz -90 deg; joints [13.301, -90.34, 134.708, -161.024, 45.01, 166.769]
  MoveL 3118 to (-311.74, 17.31, -13.97) mm, rotated rx -179.9 ry 0 rz -90 deg; joints [13.259, -90.196, 134.574, -161.085, 45.01, 166.814]
  MoveL 3119 to (-312.76, 17.24, -15.91) mm, rotated rx -179.9 ry 0 rz -90 deg; joints [13.18, -90.08, 134.467, -161.197, 45.001, 166.894]
  MoveL 3120 to (-314.4, 17.16, -17.35) mm, rotated rx -179.9 ry 0 rz -90 deg; joints [13.073, -90.005, 134.402, -161.346, 44.985, 167]
  MoveL 3121 to (-316.44, 17.08, -18.12) mm, rotated rx -179.9 ry 0 rz -90 deg; joints [12.954, -89.982, 134.386, -161.514, 44.965, 167.118]
  MoveL 3122 to (-318.63, 17.01, -18.11) mm, rotated rx -179.9 ry 0 rz -90 deg; joints [12.836, -90.012, 134.423, -161.678, 44.946, 167.234]
  MoveL 3123 to (-320.67, 16.93, -17.32) mm, rotated rx -179.9 ry 0 rz -90 deg; joints [12.736, -90.091, 134.508, -161.818, 44.929, 167.333]
  MoveL 3124 to (-322.29, 16.85, -15.86) mm, rotated rx -179.9 ry 0 rz -90 deg; joints [12.666, -90.209, 134.631, -161.915, 44.918, 167.402]
  MoveL 3125 to (-323.28, 16.78, -13.91) mm, rotated rx -179.9 ry 0 rz -90 deg; joints [12.636, -90.35, 134.775, -161.958, 44.914, 167.432]
  MoveL 3126 to (-323.52, 16.7, -11.74) mm, rotated rx -179.9 ry 0 rz -90 deg; joints [12.65, -90.496, 134.923, -161.939, 44.919, 167.42]
  MoveL 3127 to (-322.96, 16.62, -9.62) mm, rotated rx -179.9 ry 0 rz -90 deg; joints [12.706, -90.625, 135.054, -161.862, 44.933, 167.366]
  MoveL 3128 to (-321.69, 16.55, -7.84) mm, rotated rx -179.9 ry 0 rz -90 deg; joints [12.798, -90.722, 135.153, -161.737, 44.956, 167.28]
  MoveL 3129 to (-319.87, 16.47, -6.64) mm, rotated rx -179.9 ry 0 rz -90 deg; joints [12.912, -90.772, 135.207, -161.58, 44.985, 167.171]
  MoveL 3130 to (-317.74, 16.39, -6.16) mm, rotated rx -179.9 ry 0 rz -90 deg; joints [13.034, -90.768, 135.208, -161.414, 45.017, 167.057]
  MoveL 3131 to (-315.57, 16.31, -6.47) mm, rotated rx -179.9 ry 0 rz -90 deg; joints [13.148, -90.711, 135.157, -161.26, 45.05, 166.951]
  MoveL 3132 to (-313.66, 16.24, -7.53) mm, rotated rx -179.9 ry 0 rz -90 deg; joints [13.238, -90.606, 135.062, -161.139, 45.079, 166.869]
  MoveL 3133 to (-312.26, 16.16, -9.21) mm, rotated rx -179.9 ry 0 rz -90 deg; joints [13.293, -90.469, 134.935, -161.067, 45.101, 166.822]
  MoveL 3134 to (-311.54, 16.08, -11.27) mm, rotated rx -179.9 ry 0 rz -90 deg; joints [13.305, -90.317, 134.793, -161.053, 45.114, 166.815]
  MoveL 3135 to (-311.61, 16.01, -13.46) mm, rotated rx -179.9 ry 0 rz -90 deg; joints [13.273, -90.169, 134.655, -161.1, 45.116, 166.85]
  MoveL 3136 to (-312.45, 15.93, -15.48) mm, rotated rx -179.9 ry 0 rz -90 deg; joints [13.202, -90.045, 134.54, -161.201, 45.109, 166.922]
  MoveL 3137 to (-313.95, 15.85, -17.06) mm, rotated rx -179.9 ry 0 rz -90 deg; joints [13.101, -89.959, 134.464, -161.342, 45.094, 167.022]
  MoveL 3138 to (-315.92, 15.78, -18.01) mm, rotated rx -179.9 ry 0 rz -90 deg; joints [12.983, -89.923, 134.436, -161.507, 45.075, 167.138]
  MoveL 3139 to (-318.1, 15.7, -18.19) mm, rotated rx -179.9 ry 0 rz -90 deg; joints [12.864, -89.94, 134.46, -161.674, 45.055, 167.256]
  MoveL 3140 to (-320.2, 15.62, -17.58) mm, rotated rx -179.9 ry 0 rz -90 deg; joints [12.758, -90.008, 134.535, -161.821, 45.038, 167.36]
  MoveL 3141 to (-321.95, 15.55, -16.26) mm, rotated rx -179.9 ry 0 rz -90 deg; joints [12.68, -90.118, 134.65, -161.93, 45.025, 167.436]
  MoveL 3142 to (-323.11, 15.47, -14.41) mm, rotated rx -179.9 ry 0 rz -90 deg; joints [12.64, -90.255, 134.79, -161.987, 45.02, 167.477]
  MoveL 3143 to (-323.54, 15.39, -12.27) mm, rotated rx -179.9 ry 0 rz -90 deg; joints [12.643, -90.401, 134.939, -161.983, 45.023, 167.475]
  MoveL 3144 to (-323.17, 15.32, -10.11) mm, rotated rx -179.9 ry 0 rz -90 deg; joints [12.69, -90.536, 135.076, -161.92, 45.035, 167.431]
  MoveL 3145 to (-322.06, 15.24, -8.23) mm, rotated rx -179.9 ry 0 rz -90 deg; joints [12.774, -90.642, 135.184, -161.805, 45.056, 167.352]
  MoveL 3146 to (-320.35, 15.16, -6.86) mm, rotated rx -179.9 ry 0 rz -90 deg; joints [12.884, -90.704, 135.249, -161.654, 45.083, 167.248]
  MoveL 3147 to (-318.27, 15.09, -6.2) mm, rotated rx -179.9 ry 0 rz -90 deg; joints [13.005, -90.714, 135.264, -161.488, 45.115, 167.134]
  MoveL 3148 to (-316.08, 15.01, -6.32) mm, rotated rx -179.9 ry 0 rz -90 deg; joints [13.123, -90.669, 135.225, -161.329, 45.148, 167.025]
  MoveL 3149 to (-314.09, 14.93, -7.21) mm, rotated rx -179.9 ry 0 rz -90 deg; joints [13.22, -90.575, 135.139, -161.199, 45.178, 166.936]
  MoveL 3150 to (-312.54, 14.86, -8.76) mm, rotated rx -179.9 ry 0 rz -90 deg; joints [13.284, -90.444, 135.018, -161.114, 45.202, 166.88]
  MoveL 3151 to (-311.64, 14.78, -10.75) mm, rotated rx -179.9 ry 0 rz -90 deg; joints [13.307, -90.294, 134.878, -161.086, 45.216, 166.863]
  MoveL 3152 to (-311.52, 14.7, -12.94) mm, rotated rx -179.9 ry 0 rz -90 deg; joints [13.285, -90.143, 134.738, -161.118, 45.221, 166.888]
  MoveL 3153 to (-312.18, 14.63, -15.02) mm, rotated rx -179.9 ry 0 rz -90 deg; joints [13.223, -90.012, 134.616, -161.207, 45.216, 166.951]
  MoveL 3154 to (-313.54, 14.55, -16.73) mm, rotated rx -179.9 ry 0 rz -90 deg; joints [13.128, -89.915, 134.528, -161.34, 45.203, 167.045]
  MoveL 3155 to (-315.42, 14.47, -17.85) mm, rotated rx -179.9 ry 0 rz -90 deg; joints [13.013, -89.867, 134.488, -161.501, 45.185, 167.159]
  MoveL 3156 to (-317.57, 14.4, -18.22) mm, rotated rx -179.9 ry 0 rz -90 deg; joints [12.893, -89.871, 134.5, -161.668, 45.165, 167.277]
  MoveL 3157 to (-319.72, 14.32, -17.8) mm, rotated rx -179.9 ry 0 rz -90 deg; joints [12.782, -89.927, 134.563, -161.822, 45.146, 167.385]
  MoveL 3158 to (-321.57, 14.24, -16.64) mm, rotated rx -179.9 ry 0 rz -90 deg; joints [12.696, -90.028, 134.669, -161.942, 45.133, 167.469]
  MoveL 3159 to (-322.89, 14.17, -14.89) mm, rotated rx -179.9 ry 0 rz -90 deg; joints [12.647, -90.16, 134.805, -162.012, 45.126, 167.518]
  MoveL 3160 to (-323.51, 14.09, -12.8) mm, rotated rx -179.9 ry 0 rz -90 deg; joints [12.639, -90.306, 134.954, -162.023, 45.127, 167.527]
  MoveL 3161 to (-323.33, 14.01, -10.62) mm, rotated rx -179.9 ry 0 rz -90 deg; joints [12.675, -90.445, 135.096, -161.974, 45.137, 167.493]
  MoveL 3162 to (-322.39, 13.93, -8.64) mm, rotated rx -179.9 ry 0 rz -90 deg; joints [12.751, -90.56, 135.212, -161.87, 45.156, 167.422]
  MoveL 3163 to (-320.8, 13.86, -7.13) mm, rotated rx -179.9 ry 0 rz -90 deg; joints [12.856, -90.633, 135.289, -161.727, 45.182, 167.323]
  MoveL 3164 to (-318.79, 13.78, -6.29) mm, rotated rx -179.9 ry 0 rz -90 deg; joints [12.976, -90.656, 135.316, -161.563, 45.213, 167.211]
  MoveL 3165 to (-316.6, 13.7, -6.22) mm, rotated rx -179.9 ry 0 rz -90 deg; joints [13.096, -90.624, 135.29, -161.4, 45.246, 167.1]
  MoveL 3166 to (-314.54, 13.63, -6.93) mm, rotated rx -179.9 ry 0 rz -90 deg; joints [13.199, -90.541, 135.215, -161.261, 45.277, 167.005]
  MoveL 3167 to (-312.86, 13.55, -8.34) mm, rotated rx -179.9 ry 0 rz -90 deg; joints [13.272, -90.418, 135.101, -161.164, 45.302, 166.94]
  MoveL 3168 to (-311.79, 13.47, -10.24) mm, rotated rx -179.9 ry 0 rz -90 deg; joints [13.306, -90.271, 134.963, -161.122, 45.319, 166.913]
  MoveL 3169 to (-311.48, 13.4, -12.41) mm, rotated rx -179.9 ry 0 rz -90 deg; joints [13.295, -90.118, 134.821, -161.14, 45.326, 166.928]
  MoveL 3170 to (-311.95, 13.32, -14.54) mm, rotated rx -179.9 ry 0 rz -90 deg; joints [13.242, -89.981, 134.693, -161.215, 45.323, 166.982]
  MoveL 3171 to (-313.16, 13.24, -16.37) mm, rotated rx -179.9 ry 0 rz -90 deg; joints [13.154, -89.875, 134.596, -161.339, 45.311, 167.07]
  MoveL 3172 to (-314.93, 13.17, -17.64) mm, rotated rx -179.9 ry 0 rz -90 deg; joints [13.042, -89.813, 134.543, -161.494, 45.294, 167.179]
  MoveL 3173 to (-317.04, 13.09, -18.2) mm, rotated rx -179.9 ry 0 rz -90 deg; joints [12.922, -89.805, 134.542, -161.662, 45.275, 167.297]
  MoveL 3174 to (-319.22, 13.01, -17.97) mm, rotated rx -179.9 ry 0 rz -90 deg; joints [12.808, -89.849, 134.594, -161.821, 45.256, 167.409]
  MoveL 3175 to (-321.17, 12.94, -16.98) mm, rotated rx -179.9 ry 0 rz -90 deg; joints [12.715, -89.94, 134.691, -161.95, 45.241, 167.499]
  MoveL 3176 to (-322.63, 12.86, -15.36) mm, rotated rx -179.9 ry 0 rz -90 deg; joints [12.655, -90.066, 134.821, -162.033, 45.232, 167.558]
  MoveL 3177 to (-323.43, 12.78, -13.32) mm, rotated rx -179.9 ry 0 rz -90 deg; joints [12.637, -90.21, 134.969, -162.059, 45.232, 167.577]
  MoveL 3178 to (-323.44, 12.71, -11.13) mm, rotated rx -179.9 ry 0 rz -90 deg; joints [12.663, -90.352, 135.114, -162.024, 45.24, 167.553]
  MoveL 3179 to (-322.68, 12.63, -9.09) mm, rotated rx -179.9 ry 0 rz -90 deg; joints [12.73, -90.474, 135.238, -161.933, 45.257, 167.49]
  MoveL 3180 to (-321.23, 12.55, -7.44) mm, rotated rx -179.9 ry 0 rz -90 deg; joints [12.829, -90.559, 135.325, -161.798, 45.281, 167.398]
  MoveL 3181 to (-319.3, 12.48, -6.43) mm, rotated rx -179.9 ry 0 rz -90 deg; joints [12.947, -90.595, 135.365, -161.637, 45.311, 167.287]
  MoveL 3182 to (-317.13, 12.4, -6.16) mm, rotated rx -179.9 ry 0 rz -90 deg; joints [13.069, -90.576, 135.352, -161.473, 45.344, 167.175]
  MoveL 3183 to (-315.01, 12.32, -6.69) mm, rotated rx -179.9 ry 0 rz -90 deg; joints [13.177, -90.504, 135.287, -161.326, 45.375, 167.075]
  MoveL 3184 to (-313.21, 12.25, -7.94) mm, rotated rx -179.9 ry 0 rz -90 deg; joints [13.259, -90.389, 135.182, -161.218, 45.402, 167.003]
  MoveL 3185 to (-311.98, 12.17, -9.75) mm, rotated rx -179.9 ry 0 rz -90 deg; joints [13.302, -90.247, 135.048, -161.162, 45.421, 166.966]
  MoveL 3186 to (-311.48, 12.09, -11.88) mm, rotated rx -179.9 ry 0 rz -90 deg; joints [13.302, -90.094, 134.905, -161.165, 45.43, 166.97]
  MoveL 3187 to (-311.77, 12.02, -14.04) mm, rotated rx -179.9 ry 0 rz -90 deg; joints [13.259, -89.951, 134.772, -161.227, 45.429, 167.015]
  MoveL 3188 to (-312.8, 11.94, -15.97) mm, rotated rx -179.9 ry 0 rz -90 deg; joints [13.178, -89.836, 134.666, -161.34, 45.42, 167.095]
  MoveL 3189 to (-314.46, 11.86, -17.39) mm, rotated rx -179.9 ry 0 rz -90 deg; joints [13.071, -89.763, 134.602, -161.489, 45.404, 167.2]
  MoveL 3190 to (-316.52, 11.79, -18.14) mm, rotated rx -179.9 ry 0 rz -90 deg; joints [12.951, -89.742, 134.588, -161.655, 45.384, 167.317]
  MoveL 3191 to (-318.7, 11.71, -18.1) mm, rotated rx -179.9 ry 0 rz -90 deg; joints [12.834, -89.773, 134.627, -161.818, 45.365, 167.431]
  MoveL 3192 to (-320.73, 11.63, -17.28) mm, rotated rx -179.9 ry 0 rz -90 deg; joints [12.735, -89.854, 134.714, -161.956, 45.349, 167.528]
  MoveL 3193 to (-322.34, 11.55, -15.79) mm, rotated rx -179.9 ry 0 rz -90 deg; joints [12.667, -89.973, 134.838, -162.051, 45.339, 167.595]
  MoveL 3194 to (-323.31, 11.48, -13.84) mm, rotated rx -179.9 ry 0 rz -90 deg; joints [12.638, -90.114, 134.983, -162.092, 45.337, 167.623]
  MoveL 3195 to (-323.51, 11.4, -11.66) mm, rotated rx -179.9 ry 0 rz -90 deg; joints [12.654, -90.258, 135.13, -162.071, 45.343, 167.61]
  MoveL 3196 to (-322.93, 11.32, -9.55) mm, rotated rx -179.9 ry 0 rz -90 deg; joints [12.711, -90.387, 135.261, -161.993, 45.358, 167.557]
  MoveL 3197 to (-321.64, 11.25, -7.79) mm, rotated rx -179.9 ry 0 rz -90 deg; joints [12.804, -90.482, 135.359, -161.867, 45.381, 167.47]
  MoveL 3198 to (-319.8, 11.17, -6.61) mm, rotated rx -179.9 ry 0 rz -90 deg; joints [12.918, -90.53, 135.411, -161.711, 45.41, 167.363]
  MoveL 3199 to (-317.66, 11.09, -6.15) mm, rotated rx -179.9 ry 0 rz -90 deg; joints [13.041, -90.524, 135.41, -161.546, 45.442, 167.25]
  MoveL 3200 to (-315.5, 11.02, -6.49) mm, rotated rx -179.9 ry 0 rz -90 deg; joints [13.154, -90.465, 135.358, -161.393, 45.474, 167.147]
  MoveL 3201 to (-313.6, 10.94, -7.58) mm, rotated rx -179.9 ry 0 rz -90 deg; joints [13.243, -90.359, 135.261, -161.274, 45.502, 167.067]
  MoveL 3202 to (-312.22, 10.86, -9.27) mm, rotated rx -179.9 ry 0 rz -90 deg; joints [13.296, -90.222, 135.132, -161.204, 45.523, 167.021]
  MoveL 3203 to (-311.53, 10.79, -11.35) mm, rotated rx -179.9 ry 0 rz -90 deg; joints [13.307, -90.07, 134.99, -161.193, 45.534, 167.015]
  MoveL 3204 to (-311.62, 10.71, -13.53) mm, rotated rx -179.9 ry 0 rz -90 deg; joints [13.274, -89.923, 134.852, -161.241, 45.536, 167.051]
  MoveL 3205 to (-312.49, 10.63, -15.54) mm, rotated rx -179.9 ry 0 rz -90 deg; joints [13.201, -89.8, 134.738, -161.343, 45.528, 167.123]
  MoveL 3206 to (-314.02, 10.56, -17.11) mm, rotated rx -179.9 ry 0 rz -90 deg; joints [13.099, -89.716, 134.663, -161.484, 45.513, 167.222]
  MoveL 3207 to (-316, 10.48, -18.03) mm, rotated rx -179.9 ry 0 rz -90 deg; joints [12.981, -89.681, 134.636, -161.648, 45.494, 167.337]
  MoveL 3208 to (-318.18, 10.4, -18.18) mm, rotated rx -179.9 ry 0 rz -90 deg; joints [12.862, -89.7, 134.663, -161.814, 45.475, 167.453]
  MoveL 3209 to (-320.27, 10.33, -17.54) mm, rotated rx -179.9 ry 0 rz -90 deg; joints [12.757, -89.77, 134.739, -161.959, 45.458, 167.554]
  MoveL 3210 to (-322, 10.25, -16.21) mm, rotated rx -179.9 ry 0 rz -90 deg; joints [12.68, -89.881, 134.855, -162.066, 45.447, 167.629]
  MoveL 3211 to (-323.14, 10.17, -14.34) mm, rotated rx -179.9 ry 0 rz -90 deg; joints [12.642, -90.018, 134.997, -162.12, 45.442, 167.668]
  MoveL 3212 to (-323.54, 10.1, -12.19) mm, rotated rx -179.9 ry 0 rz -90 deg; joints [12.646, -90.163, 135.146, -162.115, 45.447, 167.665]
  MoveL 3213 to (-323.14, 10.02, -10.04) mm, rotated rx -179.9 ry 0 rz -90 deg; joints [12.694, -90.297, 135.283, -162.05, 45.46, 167.621]
  MoveL 3214 to (-322.01, 9.94, -8.17) mm, rotated rx -179.9 ry 0 rz -90 deg; joints [12.779, -90.402, 135.39, -161.935, 45.481, 167.542]
  MoveL 3215 to (-320.28, 9.87, -6.83) mm, rotated rx -179.9 ry 0 rz -90 deg; joints [12.89, -90.462, 135.453, -161.784, 45.509, 167.439]
  MoveL 3216 to (-318.19, 9.79, -6.19) mm, rotated rx -179.9 ry 0 rz -90 deg; joints [13.012, -90.469, 135.466, -161.619, 45.54, 167.326]
  MoveL 3217 to (-316.01, 9.71, -6.34) mm, rotated rx -179.9 ry 0 rz -90 deg; joints [13.129, -90.422, 135.425, -161.462, 45.572, 167.219]
  MoveL 3218 to (-314.02, 9.64, -7.26) mm, rotated rx -179.9 ry 0 rz -90 deg; joints [13.225, -90.327, 135.338, -161.333, 45.602, 167.133]
  MoveL 3219 to (-312.5, 9.56, -8.82) mm, rotated rx -179.9 ry 0 rz -90 deg; joints [13.287, -90.196, 135.215, -161.251, 45.624, 167.078]
  MoveL 3220 to (-311.63, 9.48, -10.83) mm, rotated rx -179.9 ry 0 rz -90 deg; joints [13.309, -90.046, 135.074, -161.225, 45.638, 167.062]
  MoveL 3221 to (-311.53, 9.41, -13.01) mm, rotated rx -179.9 ry 0 rz -90 deg; joints [13.286, -89.896, 134.934, -161.259, 45.641, 167.088]
  MoveL 3222 to (-312.22, 9.33, -15.09) mm, rotated rx -179.9 ry 0 rz -90 deg; joints [13.222, -89.765, 134.813, -161.348, 45.636, 167.151]
  MoveL 3223 to (-313.6, 9.25, -16.78) mm, rotated rx -179.9 ry 0 rz -90 deg; joints [13.127, -89.671, 134.727, -161.481, 45.622, 167.245]
  MoveL 3224 to (-315.49, 9.18, -17.87) mm, rotated rx -179.9 ry 0 rz -90 deg; joints [13.011, -89.624, 134.688, -161.641, 45.604, 167.357]
  MoveL 3225 to (-317.65, 9.1, -18.22) mm, rotated rx -179.9 ry 0 rz -90 deg; joints [12.89, -89.63, 134.702, -161.808, 45.585, 167.473]
  MoveL 3226 to (-319.79, 9.02, -17.77) mm, rotated rx -179.9 ry 0 rz -90 deg; joints [12.781, -89.688, 134.766, -161.96, 45.567, 167.58]
  MoveL 3227 to (-321.63, 8.94, -16.58) mm, rotated rx -179.9 ry 0 rz -90 deg; joints [12.696, -89.79, 134.874, -162.078, 45.554, 167.662]
  MoveL 3228 to (-322.93, 8.87, -14.82) mm, rotated rx -179.9 ry 0 rz -90 deg; joints [12.648, -89.922, 135.012, -162.145, 45.549, 167.71]
  MoveL 3229 to (-323.51, 8.79, -12.72) mm, rotated rx -179.9 ry 0 rz -90 deg; joints [12.642, -90.067, 135.16, -162.155, 45.551, 167.717]
  MoveL 3230 to (-323.31, 8.71, -10.54) mm, rotated rx -179.9 ry 0 rz -90 deg; joints [12.68, -90.206, 135.302, -162.104, 45.562, 167.682]
  MoveL 3231 to (-322.34, 8.64, -8.58) mm, rotated rx -179.9 ry 0 rz -90 deg; joints [12.756, -90.319, 135.418, -162, 45.581, 167.611]
  MoveL 3232 to (-320.74, 8.56, -7.09) mm, rotated rx -179.9 ry 0 rz -90 deg; joints [12.862, -90.39, 135.493, -161.856, 45.608, 167.513]
  MoveL 3233 to (-318.71, 8.48, -6.27) mm, rotated rx -179.9 ry 0 rz -90 deg; joints [12.983, -90.411, 135.518, -161.693, 45.639, 167.402]
  MoveL 3234 to (-316.53, 8.41, -6.23) mm, rotated rx -179.9 ry 0 rz -90 deg; joints [13.102, -90.377, 135.49, -161.532, 45.671, 167.293]
  MoveL 3235 to (-314.47, 8.33, -6.97) mm, rotated rx -179.9 ry 0 rz -90 deg; joints [13.205, -90.292, 135.413, -161.395, 45.701, 167.201]
  MoveL 3236 to (-312.81, 8.25, -8.4) mm, rotated rx -179.9 ry 0 rz -90 deg; joints [13.276, -90.169, 135.297, -161.3, 45.725, 167.137]
  MoveL 3237 to (-311.77, 8.18, -10.32) mm, rotated rx -179.9 ry 0 rz -90 deg; joints [13.308, -90.021, 135.159, -161.26, 45.741, 167.112]
  MoveL 3238 to (-311.48, 8.1, -12.48) mm, rotated rx -179.9 ry 0 rz -90 deg; joints [13.296, -89.87, 135.017, -161.279, 45.747, 167.127]
  MoveL 3239 to (-311.98, 8.02, -14.61) mm, rotated rx -179.9 ry 0 rz -90 deg; joints [13.242, -89.733, 134.889, -161.356, 45.743, 167.182]
  MoveL 3240 to (-313.21, 7.95, -16.42) mm, rotated rx -179.9 ry 0 rz -90 deg; joints [13.153, -89.629, 134.793, -161.48, 45.731, 167.269]
  MoveL 3241 to (-315, 7.87, -17.67) mm, rotated rx -179.9 ry 0 rz -90 deg; joints [13.04, -89.569, 134.742, -161.635, 45.714, 167.377]
  MoveL 3242 to (-317.12, 7.79, -18.2) mm, rotated rx -179.9 ry 0 rz -90 deg; joints [12.92, -89.563, 134.743, -161.802, 45.695, 167.494]
  MoveL 3243 to (-319.29, 7.72, -17.95) mm, rotated rx -179.9 ry 0 rz -90 deg; joints [12.806, -89.608, 134.796, -161.959, 45.677, 167.603]
  MoveL 3244 to (-321.23, 7.64, -16.93) mm, rotated rx -179.9 ry 0 rz -90 deg; joints [12.714, -89.701, 134.895, -162.086, 45.663, 167.692]
  MoveL 3245 to (-322.68, 7.56, -15.29) mm, rotated rx -179.9 ry 0 rz -90 deg; joints [12.656, -89.827, 135.026, -162.167, 45.655, 167.749]
  MoveL 3246 to (-323.44, 7.49, -13.24) mm, rotated rx -179.9 ry 0 rz -90 deg; joints [12.64, -89.971, 135.174, -162.191, 45.656, 167.766]
  MoveL 3247 to (-323.43, 7.41, -11.06) mm, rotated rx -179.9 ry 0 rz -90 deg; joints [12.667, -90.112, 135.319, -162.154, 45.665, 167.742]
  MoveL 3248 to (-322.64, 7.33, -9.02) mm, rotated rx -179.9 ry 0 rz -90 deg; joints [12.735, -90.233, 135.443, -162.062, 45.682, 167.679]
  MoveL 3249 to (-321.17, 7.26, -7.4) mm, rotated rx -179.9 ry 0 rz -90 deg; joints [12.835, -90.316, 135.529, -161.927, 45.707, 167.587]
  MoveL 3250 to (-319.23, 7.18, -6.4) mm, rotated rx -179.9 ry 0 rz -90 deg; joints [12.954, -90.349, 135.567, -161.766, 45.737, 167.478]
  MoveL 3251 to (-317.05, 7.1, -6.17) mm, rotated rx -179.9 ry 0 rz -90 deg; joints [13.075, -90.328, 135.551, -161.603, 45.769, 167.367]
  MoveL 3252 to (-314.94, 7.03, -6.72) mm, rotated rx -179.9 ry 0 rz -90 deg; joints [13.183, -90.255, 135.485, -161.458, 45.8, 167.27]
  MoveL 3253 to (-313.16, 6.95, -8) mm, rotated rx -179.9 ry 0 rz -90 deg; joints [13.263, -90.14, 135.378, -161.352, 45.826, 167.199]
  MoveL 3254 to (-311.95, 6.87, -9.82) mm, rotated rx -179.9 ry 0 rz -90 deg; joints [13.305, -89.996, 135.244, -161.298, 45.844, 167.164]
  MoveL 3255 to (-311.48, 6.8, -11.95) mm, rotated rx -179.9 ry 0 rz -90 deg; joints [13.303, -89.844, 135.1, -161.303, 45.852, 167.169]
  MoveL 3256 to (-311.79, 6.72, -14.12) mm, rotated rx -179.9 ry 0 rz -90 deg; joints [13.259, -89.702, 134.967, -161.366, 45.85, 167.215]
  MoveL 3257 to (-312.85, 6.64, -16.03) mm, rotated rx -179.9 ry 0 rz -90 deg; joints [13.177, -89.589, 134.862, -161.48, 45.84, 167.294]
  MoveL 3258 to (-314.53, 6.56, -17.43) mm, rotated rx -179.9 ry 0 rz -90 deg; joints [13.069, -89.518, 134.799, -161.629, 45.824, 167.398]
  MoveL 3259 to (-316.59, 6.49, -18.15) mm, rotated rx -179.9 ry 0 rz -90 deg; joints [12.949, -89.498, 134.788, -161.794, 45.805, 167.514]
  MoveL 3260 to (-318.78, 6.41, -18.08) mm, rotated rx -179.9 ry 0 rz -90 deg; joints [12.832, -89.531, 134.828, -161.956, 45.786, 167.626]
  MoveL 3261 to (-320.8, 6.33, -17.24) mm, rotated rx -179.9 ry 0 rz -90 deg; joints [12.734, -89.613, 134.917, -162.092, 45.771, 167.72]
  MoveL 3262 to (-322.38, 6.26, -15.73) mm, rotated rx -179.9 ry 0 rz -90 deg; joints [12.667, -89.733, 135.042, -162.185, 45.762, 167.786]
  MoveL 3263 to (-323.33, 6.18, -13.76) mm, rotated rx -179.9 ry 0 rz -90 deg; joints [12.64, -89.874, 135.188, -162.223, 45.761, 167.813]
  MoveL 3264 to (-323.51, 6.1, -11.58) mm, rotated rx -179.9 ry 0 rz -90 deg; joints [12.657, -90.018, 135.336, -162.201, 45.768, 167.798]
  MoveL 3265 to (-322.9, 6.03, -9.48) mm, rotated rx -179.9 ry 0 rz -90 deg; joints [12.716, -90.145, 135.466, -162.121, 45.784, 167.745]
  MoveL 3266 to (-321.58, 5.95, -7.74) mm, rotated rx -179.9 ry 0 rz -90 deg; joints [12.809, -90.238, 135.562, -161.995, 45.807, 167.659]
  MoveL 3267 to (-319.73, 5.87, -6.58) mm, rotated rx -179.9 ry 0 rz -90 deg; joints [12.925, -90.284, 135.612, -161.839, 45.836, 167.553]
  MoveL 3268 to (-317.58, 5.8, -6.15) mm, rotated rx -179.9 ry 0 rz -90 deg; joints [13.047, -90.276, 135.61, -161.675, 45.868, 167.442]
  MoveL 3269 to (-315.43, 5.72, -6.52) mm, rotated rx -179.9 ry 0 rz -90 deg; joints [13.16, -90.215, 135.556, -161.524, 45.899, 167.34]
  MoveL 3270 to (-313.54, 5.64, -7.63) mm, rotated rx -179.9 ry 0 rz -90 deg; joints [13.247, -90.109, 135.457, -161.407, 45.926, 167.262]
  MoveL 3271 to (-312.18, 5.57, -9.34) mm, rotated rx -179.9 ry 0 rz -90 deg; joints [13.299, -89.971, 135.327, -161.34, 45.946, 167.218]
  MoveL 3272 to (-311.52, 5.49, -11.43) mm, rotated rx -179.9 ry 0 rz -90 deg; joints [13.308, -89.819, 135.184, -161.33, 45.956, 167.213]
  MoveL 3273 to (-311.64, 5.41, -13.61) mm, rotated rx -179.9 ry 0 rz -90 deg; joints [13.274, -89.673, 135.047, -161.38, 45.957, 167.249]
  MoveL 3274 to (-312.53, 5.34, -15.6) mm, rotated rx -179.9 ry 0 rz -90 deg; joints [13.2, -89.551, 134.934, -161.482, 45.948, 167.321]
  MoveL 3275 to (-314.08, 5.26, -17.15) mm, rotated rx -179.9 ry 0 rz -90 deg; joints [13.098, -89.469, 134.86, -161.624, 45.933, 167.42]
  MoveL 3276 to (-316.07, 5.18, -18.05) mm, rotated rx -179.9 ry 0 rz -90 deg; joints [12.979, -89.436, 134.835, -161.787, 45.915, 167.533]
  MoveL 3277 to (-318.26, 5.11, -18.17) mm, rotated rx -179.9 ry 0 rz -90 deg; joints [12.86, -89.457, 134.863, -161.951, 45.896, 167.647]
  MoveL 3278 to (-320.34, 5.03, -17.51) mm, rotated rx -179.9 ry 0 rz -90 deg; joints [12.756, -89.528, 134.941, -162.095, 45.88, 167.747]
  MoveL 3279 to (-322.05, 4.95, -16.15) mm, rotated rx -179.9 ry 0 rz -90 deg; joints [12.68, -89.64, 135.059, -162.199, 45.87, 167.82]
  MoveL 3280 to (-323.17, 4.88, -14.27) mm, rotated rx -179.9 ry 0 rz -90 deg; joints [12.643, -89.777, 135.202, -162.251, 45.867, 167.857]
  MoveL 3281 to (-323.54, 4.8, -12.11) mm, rotated rx -179.9 ry 0 rz -90 deg; joints [12.65, -89.922, 135.351, -162.244, 45.872, 167.853]
  MoveL 3282 to (-323.11, 4.72, -9.97) mm, rotated rx -179.9 ry 0 rz -90 deg; joints [12.699, -90.055, 135.487, -162.178, 45.886, 167.808]
  MoveL 3283 to (-321.95, 4.65, -8.11) mm, rotated rx -179.9 ry 0 rz -90 deg; joints [12.785, -90.157, 135.593, -162.062, 45.907, 167.73]
  MoveL 3284 to (-320.21, 4.57, -6.79) mm, rotated rx -179.9 ry 0 rz -90 deg; joints [12.896, -90.216, 135.655, -161.912, 45.935, 167.628]
  MoveL 3285 to (-318.11, 4.49, -6.18) mm, rotated rx -179.9 ry 0 rz -90 deg; joints [13.018, -90.221, 135.665, -161.747, 45.967, 167.517]
  MoveL 3286 to (-315.93, 4.42, -6.36) mm, rotated rx -179.9 ry 0 rz -90 deg; joints [13.135, -90.172, 135.623, -161.592, 45.998, 167.412]
  MoveL 3287 to (-313.96, 4.34, -7.3) mm, rotated rx -179.9 ry 0 rz -90 deg; joints [13.23, -90.076, 135.534, -161.465, 46.026, 167.327]
  MoveL 3288 to (-312.45, 4.26, -8.89) mm, rotated rx -179.9 ry 0 rz -90 deg; joints [13.291, -89.944, 135.41, -161.385, 46.048, 167.274]
  MoveL 3289 to (-311.61, 4.18, -10.9) mm, rotated rx -179.9 ry 0 rz -90 deg; joints [13.311, -89.794, 135.268, -161.361, 46.06, 167.26]
  MoveL 3290 to (-311.54, 4.11, -13.09) mm, rotated rx -179.9 ry 0 rz -90 deg; joints [13.286, -89.645, 135.128, -161.396, 46.063, 167.286]
  MoveL 3291 to (-312.25, 4.03, -15.16) mm, rotated rx -179.9 ry 0 rz -90 deg; joints [13.222, -89.516, 135.007, -161.486, 46.057, 167.349]
  MoveL 3292 to (-313.66, 3.95, -16.83) mm, rotated rx -179.9 ry 0 rz -90 deg; joints [13.125, -89.423, 134.923, -161.62, 46.043, 167.442]
  MoveL 3293 to (-315.57, 3.88, -17.9) mm, rotated rx -179.9 ry 0 rz -90 deg; joints [13.009, -89.378, 134.885, -161.78, 46.025, 167.553]
  MoveL 3294 to (-317.73, 3.8, -18.21) mm, rotated rx -179.9 ry 0 rz -90 deg; joints [12.888, -89.386, 134.901, -161.945, 46.006, 167.668]
  MoveL 3295 to (-319.86, 3.72, -17.74) mm, rotated rx -179.9 ry 0 rz -90 deg; joints [12.779, -89.445, 134.968, -162.095, 45.989, 167.772]
